				(*571*) (*ALL 571 AND SUBS*)
					OR ((Model_ID=7)
						(*AND Part_Present1 AND Part_Present2 AND Part_Present3
						AND Part_Present4 AND Part_Present5 AND Part_Present6
						AND Part_Present7 AND NOT Part_Present8 AND NOT Part_Present9
						AND NOT Part_Present10 AND NOT Part_Present11 AND NOT Part_Present12
						AND NOT Part_Present13 AND Part_Present15 AND NOT Part_Present16 
						AND NOT Part_Present17 AND NOT Part_Present18 AND NOT Part_Present19 
						AND NOT Part_Present20 AND NOT Part_Present21 AND Part_Present22 
						AND Part_Present23 AND Part_Present24 AND NOT Part_Present25 
						AND NOT Part_Present29 
						AND NOT Part_Present30 AND NOT Part_Present31 AND NOT Part_Present32 
						AND Part_Present33 AND Part_Present34 AND Part_Present35 
						AND Part_Present36 AND Part_Present37 AND Part_Present38 
						AND NOT Part_Present39 AND NOT Part_Present40 AND NOT Part_Present41 
						AND NOT Part_Present42 AND NOT Part_Present43 AND Part_Present45
						AND Part_Present46 AND Part_Present47 AND Part_Present48
						AND Part_Present49 AND Part_Present50 AND Part_Present51
						AND NOT Part_Present52 AND NOT Part_Present53 AND NOT Part_Present54
						AND NOT Part_Present55 AND NOT Part_Present56 AND NOT Part_Present57
						AND Part_Present62 AND Part_Present63 AND Part_Present64*)

						AND Part_Present1 AND Part_Present2 AND  Part_Present3
						AND Part_Present4 AND Part_Present5 AND Part_Present6
						AND Part_Present7 AND NOT Part_Present8 AND NOT Part_Present9
						AND NOT Part_Present10 AND NOT Part_Present11 AND NOT Part_Present12
						AND NOT Part_Present13 AND NOT Part_Present14 AND Part_Present15
						AND NOT Part_Present16 AND NOT Part_Present17 AND NOT Part_Present18
						AND NOT Part_Present19 AND NOT Part_Present20 AND NOT Part_Present21
						AND Part_Present22 AND Part_Present23 AND Part_Present24
						AND NOT Part_Present25 AND NOT Part_Present26 AND NOT Part_Present27
						AND NOT Part_Present28 AND NOT Part_Present29 AND NOT Part_Present30
						AND NOT Part_Present31 AND NOT Part_Present32 AND Part_Present33
						AND Part_Present34 AND Part_Present35 AND Part_Present36
						AND Part_Present37 AND Part_Present38 AND NOT Part_Present39
						AND NOT Part_Present40 AND NOT Part_Present41 AND NOT Part_Present42 
						AND NOT Part_Present43 AND NOT Part_Present44 AND Part_Present45
						AND Part_Present46 AND Part_Present47 AND Part_Present48
						AND Part_Present49 AND Part_Present50 AND Part_Present51
						AND NOT Part_Present52 AND NOT Part_Present53 AND NOT Part_Present54
						AND NOT Part_Present55 AND NOT Part_Present56 AND NOT Part_Present57
						AND NOT Part_Present58 AND NOT Part_Present59 AND NOT Part_Present60
						AND NOT Part_Present61 AND Part_Present62 AND Part_Present63
						AND Part_Present64 AND NOT Part_Present65 AND NOT Part_Present66
						AND NOT Part_Present67 AND NOT Part_Present68 AND NOT Part_Present69
						AND NOT Part_Present70 AND NOT Part_Present71 AND NOT Part_Present72
						AND NOT Part_Present73 AND NOT Part_Present74 AND NOT Part_Present75
						AND NOT Part_Present76)			
					) OR (All_Sensors_Off AND Dry_Cycle)
					
					(*504 SUBS 1,2*)
					OR (((Model_ID=8) AND All_Sensors_On.9 AND All_Sensors_On.10)							

					(*524 SUBS 1,2*)
					OR ((Model_ID=9) AND All_Sensors_On.9 AND All_Sensors_On.10)							

					(*543 SUBS 1,2,5*)
					OR ((Model_ID=10) AND All_Sensors_On.9 AND All_Sensors_On.10 AND All_Sensors_On.13)							
							
					(*526 SUBS 1-3*)
					OR ((Model_ID=11) AND All_Sensors_On.9 AND All_Sensors_On.10 AND All_Sensors_On.11)
							
					(*526 SUBS 4 ONLY*)
					OR ((Model_ID=15) AND All_Sensors_On.12)
							
					(*526 SUBS 1-4*)
					OR ((Model_ID=19) AND All_Sensors_On.9 AND All_Sensors_On.10 AND All_Sensors_On.11 AND All_Sensors_On.12)
					
					(*536 SUBS 1-3*)
					OR ((Model_ID=12) AND All_Sensors_On.9 AND All_Sensors_On.10 AND All_Sensors_On.11)
							
					(*536 SUBS 4 ONLY*)
					OR ((Model_ID=16) AND All_Sensors_On.12)
							
					(*536 SUBS 1-4*)
					OR ((Model_ID=20) AND All_Sensors_On.9 AND All_Sensors_On.10 AND All_Sensors_On.11 AND All_Sensors_On.12)
					
					(*550 SUBS 1-3*)
					OR ((Model_ID=13) AND All_Sensors_On.9 AND All_Sensors_On.10 AND All_Sensors_On.11)
							
					(*550 SUBS 4 ONLY*)
					OR ((Model_ID=17) AND All_Sensors_On.12)
							
					(*550 SUBS 1-4*)
					OR ((Model_ID=21) AND All_Sensors_On.9 AND All_Sensors_On.10 AND All_Sensors_On.11 AND All_Sensors_On.12)
					
					(*571 SUBS 1-3*)
					OR ((Model_ID=14) AND All_Sensors_On.9 AND All_Sensors_On.10 AND All_Sensors_On.11)
							
					(*571 SUBS 4 ONLY*)
					OR ((Model_ID=18) AND All_Sensors_On.12)
							
					(*571 SUBS 1-4*)
					OR ((Model_ID=22) AND All_Sensors_On.9 AND All_Sensors_On.10 AND All_Sensors_On.11 AND All_Sensors_On.12));

	(*Sensors Required for Resetting Subs*)
	(*SUB 1 - Not Checking Sub 1,2 sensors as we are building 1-3*)
	All_Sensors_On.9:= ((*NOT Part_Present1 AND NOT Part_Present2 AND NOT  Part_Present3
						AND NOT Part_Present4 AND NOT Part_Present5 AND NOT Part_Present6
						AND NOT Part_Present7*)NOT Part_Present8 AND NOT Part_Present9
						AND NOT Part_Present10 AND NOT Part_Present11 AND NOT Part_Present12
						AND NOT Part_Present13 AND NOT Part_Present14 AND NOT Part_Present15
						AND NOT Part_Present16 AND NOT Part_Present17 AND NOT Part_Present18
						AND NOT Part_Present19 AND NOT Part_Present20 (*AND NOT Part_Present21*)
						AND NOT Part_Present22 AND NOT Part_Present23 AND NOT Part_Present24
						AND NOT Part_Present25 AND NOT Part_Present26 AND NOT Part_Present27
						AND NOT Part_Present28 AND NOT Part_Present29 AND NOT Part_Present30
						AND NOT Part_Present31 AND NOT Part_Present32 AND NOT Part_Present33
						AND NOT Part_Present34 AND NOT Part_Present35 AND NOT Part_Present36
						AND NOT Part_Present37 AND NOT Part_Present38 AND NOT Part_Present39
						AND NOT Part_Present40 AND NOT Part_Present41 AND NOT Part_Present42 
						AND NOT Part_Present43 AND NOT Part_Present44 (*AND NOT Part_Present45
						AND NOT Part_Present46 AND NOT Part_Present47 AND NOT Part_Present48
						AND NOT Part_Present49 AND NOT Part_Present50 AND NOT Part_Present51*)
						AND NOT Part_Present52 AND NOT Part_Present53 AND NOT Part_Present54
						AND NOT Part_Present55 AND NOT Part_Present56 AND NOT Part_Present57
						AND NOT Part_Present58 AND NOT Part_Present59 AND NOT Part_Present60
						AND NOT Part_Present61 AND NOT Part_Present62 AND NOT Part_Present63
						AND NOT Part_Present64 AND NOT Part_Present65 AND NOT Part_Present66
						AND NOT Part_Present67 AND NOT Part_Present68 AND NOT Part_Present69
						AND NOT Part_Present70 AND NOT Part_Present71 AND NOT Part_Present72
						(*AND NOT Part_Present73*) AND NOT Part_Present74 (*AND NOT Part_Present75*)
						AND NOT Part_Present76)
					  AND
						(((Model_ID=8) AND( NOT Part_Present1 AND NOT Part_Present2 AND NOT Part_Present3
									   AND NOT Part_Present4 AND NOT Part_Present5 AND Part_Present6
									   AND Part_Present7))
										
					  OR ((Model_ID=9) AND( NOT Part_Present1 AND NOT Part_Present2 AND NOT Part_Present3
									   AND NOT Part_Present4 AND Part_Present5 AND Part_Present6
									   AND Part_Present7))
										
					  OR ((Model_ID=10) AND( NOT Part_Present1 AND NOT Part_Present2 AND NOT Part_Present3
									    AND NOT Part_Present4 AND NOT Part_Present5 AND NOT Part_Present6
									    AND Part_Present7))
									   
					  OR ((Model_ID=11) AND(Part_Present1 AND NOT Part_Present2 AND NOT Part_Present3
									    AND NOT Part_Present4 AND Part_Present5 AND Part_Present6
									    AND Part_Present7))
									   
					  OR ((Model_ID=12) AND(Part_Present1 AND NOT Part_Present2 AND NOT Part_Present3
									    AND Part_Present4 AND Part_Present5 AND Part_Present6
									    AND Part_Present7))
									   
					  OR ((Model_ID=13) AND(Part_Present1 AND NOT Part_Present2 AND Part_Present3
									    AND Part_Present4 AND Part_Present5 AND Part_Present6
									    AND Part_Present7))
									   
					  OR ((Model_ID=14) AND(Part_Present1 AND Part_Present2 AND Part_Present3
									    AND Part_Present4 AND Part_Present5 AND Part_Present6
									    AND Part_Present7)))

						OR (All_Sensors_Off AND Dry_Cycle);

	(*SUB 2 - Not Checking Sub 1,2 as we are building 1-3*)
	All_Sensors_On.10:= ((*NOT Part_Present1 AND NOT Part_Present2 AND NOT  Part_Present3
						AND NOT Part_Present4 AND NOT Part_Present5 AND NOT Part_Present6
						AND NOT Part_Present7*)NOT Part_Present8 AND NOT Part_Present9
						AND NOT Part_Present10 AND NOT Part_Present11 AND NOT Part_Present12
						AND NOT Part_Present13 AND NOT Part_Present14 AND NOT Part_Present15
						AND NOT Part_Present16 AND NOT Part_Present17 AND NOT Part_Present18
						AND NOT Part_Present19 AND NOT Part_Present20 (*AND NOT Part_Present21*)
						AND NOT Part_Present22 AND NOT Part_Present23 AND NOT Part_Present24
						AND NOT Part_Present25 AND NOT Part_Present26 AND NOT Part_Present27
						AND NOT Part_Present28 AND NOT Part_Present29 AND NOT Part_Present30
						AND NOT Part_Present31 AND NOT Part_Present32 AND NOT Part_Present33
						AND NOT Part_Present34 AND NOT Part_Present35 AND NOT Part_Present36
						AND NOT Part_Present37 AND NOT Part_Present38 AND NOT Part_Present39
						AND NOT Part_Present40 AND NOT Part_Present41 AND NOT Part_Present42 
						AND NOT Part_Present43 AND NOT Part_Present44 (*AND NOT Part_Present45
						AND NOT Part_Present46 AND NOT Part_Present47 AND NOT Part_Present48
						AND NOT Part_Present49 AND NOT Part_Present50 AND NOT Part_Present51*)
						AND NOT Part_Present52 AND NOT Part_Present53 AND NOT Part_Present54
						AND NOT Part_Present55 AND NOT Part_Present56 AND NOT Part_Present57
						AND NOT Part_Present58 AND NOT Part_Present59 AND NOT Part_Present60
						AND NOT Part_Present61 AND NOT Part_Present62 AND NOT Part_Present63
						AND NOT Part_Present64 AND NOT Part_Present65 AND NOT Part_Present66
						AND NOT Part_Present67 AND NOT Part_Present68 AND NOT Part_Present69
						AND NOT Part_Present70 AND NOT Part_Present71 AND NOT Part_Present72
						(*AND NOT Part_Present73*) AND NOT Part_Present74 (*AND NOT Part_Present75*)
						AND NOT Part_Present76)
						AND
						(((Model_ID=8) AND( NOT Part_Present45
											AND NOT Part_Present46 AND NOT Part_Present47 AND NOT Part_Present48
											AND NOT Part_Present49 AND Part_Present50 AND Part_Present51))
										
					  OR ((Model_ID=9) AND( NOT Part_Present45
											AND NOT Part_Present46 AND NOT Part_Present47 AND NOT Part_Present48
											AND Part_Present49 AND Part_Present50 AND Part_Present51))
										
					  OR ((Model_ID=10) AND( NOT Part_Present45
											AND NOT Part_Present46 AND NOT Part_Present47 AND NOT Part_Present48
											AND NOT Part_Present49 AND NOT Part_Present50 AND Part_Present51))
									   
					  OR ((Model_ID=11) AND(NOT Part_Present45
											AND NOT Part_Present46 AND NOT Part_Present47 AND Part_Present48
											AND Part_Present49 AND Part_Present50 AND Part_Present51))
									   
					  OR ((Model_ID=12) AND(NOT Part_Present45
											AND NOT Part_Present46 AND Part_Present47 AND Part_Present48
											AND Part_Present49 AND Part_Present50 AND Part_Present51))
									   
					  OR ((Model_ID=13) AND(NOT Part_Present45
											AND Part_Present46 AND Part_Present47 AND Part_Present48
											AND Part_Present49 AND Part_Present50 AND Part_Present51))
									   
					  OR ((Model_ID=14) AND(Part_Present45
											AND Part_Present46 AND Part_Present47 AND Part_Present48
											AND Part_Present49 AND Part_Present50 AND Part_Present51)))

			 OR (All_Sensors_Off AND Dry_Cycle);

	(*SUB 3 - Not Checking Sub 1,2 as we are building 1-3*)
	All_Sensors_On.11:=((*NOT Part_Present1 AND NOT Part_Present2 AND NOT  Part_Present3
						AND NOT Part_Present4 AND NOT Part_Present5 AND NOT Part_Present6
						AND NOT Part_Present7*)NOT Part_Present8 AND NOT Part_Present9
						AND NOT Part_Present10 AND NOT Part_Present11 AND NOT Part_Present12
						AND NOT Part_Present13 AND NOT Part_Present14 AND NOT Part_Present15
						AND NOT Part_Present16 AND NOT Part_Present17 AND NOT Part_Present18
						AND NOT Part_Present19 AND NOT Part_Present20 (*AND NOT Part_Present21*)
						AND NOT Part_Present22 AND NOT Part_Present23 AND NOT Part_Present24
						AND NOT Part_Present25 AND NOT Part_Present26 AND NOT Part_Present27
						AND NOT Part_Present28 AND NOT Part_Present29 AND NOT Part_Present30
						AND NOT Part_Present31 AND NOT Part_Present32 AND NOT Part_Present33
						AND NOT Part_Present34 AND NOT Part_Present35 AND NOT Part_Present36
						AND NOT Part_Present37 AND NOT Part_Present38 AND NOT Part_Present39
						AND NOT Part_Present40 AND NOT Part_Present41 AND NOT Part_Present42 
						AND NOT Part_Present43 AND NOT Part_Present44 (*AND NOT Part_Present45
						AND NOT Part_Present46 AND NOT Part_Present47 AND NOT Part_Present48
						AND NOT Part_Present49 AND NOT Part_Present50 AND NOT Part_Present51*)
						AND NOT Part_Present52 AND NOT Part_Present53 AND NOT Part_Present54
						AND NOT Part_Present55 AND NOT Part_Present56 AND NOT Part_Present57
						AND NOT Part_Present58 AND NOT Part_Present59 AND NOT Part_Present60
						AND NOT Part_Present61 AND NOT Part_Present62 AND NOT Part_Present63
						AND NOT Part_Present64 AND NOT Part_Present65 AND NOT Part_Present66
						AND NOT Part_Present67 AND NOT Part_Present68 AND NOT Part_Present69
						AND NOT Part_Present70 AND NOT Part_Present71 AND NOT Part_Present72
						(*AND NOT Part_Present73*) AND NOT Part_Present74 (*AND NOT Part_Present75*)
						AND NOT Part_Present76)
						AND
						(((Model_ID=11) AND(Part_Present21))
									   
					  OR ((Model_ID=12) AND(Part_Present21))
									   
					  OR ((Model_ID=13) AND(Part_Present21))
									   
					  OR ((Model_ID=14) AND(Part_Present21)))

		 	OR (All_Sensors_Off AND Dry_Cycle);

	(*SUB 4 - Checking only SUB 4 Sensors*)
	All_Sensors_On.12:=(NOT Part_Present1 AND NOT Part_Present2 AND NOT  Part_Present3
						AND NOT Part_Present4 AND NOT Part_Present5 AND NOT Part_Present6
						AND NOT Part_Present7  AND NOT Part_Present8 AND NOT Part_Present9
						AND NOT Part_Present10 AND NOT Part_Present11 AND NOT Part_Present12
						AND NOT Part_Present13 AND NOT Part_Present14 AND NOT Part_Present15
						AND NOT Part_Present16 AND NOT Part_Present17 AND NOT Part_Present18
						AND NOT Part_Present19 AND NOT Part_Present20 AND NOT Part_Present21
						AND NOT Part_Present22 AND NOT Part_Present23 AND NOT Part_Present24
						AND NOT Part_Present25 AND NOT Part_Present26 AND NOT Part_Present27
						AND NOT Part_Present28 AND NOT Part_Present29 AND NOT Part_Present30
						AND NOT Part_Present31 AND NOT Part_Present32 (*AND NOT Part_Present33
						AND NOT Part_Present34 AND NOT Part_Present35 AND NOT Part_Present36
						AND NOT Part_Present37*) AND NOT Part_Present38 AND NOT Part_Present39
						AND NOT Part_Present40 AND NOT Part_Present41 AND NOT Part_Present42 
						AND NOT Part_Present43 AND NOT Part_Present44 AND NOT Part_Present45
						AND NOT Part_Present46 AND NOT Part_Present47 AND NOT Part_Present48
						AND NOT Part_Present49 AND NOT Part_Present50 AND NOT Part_Present51
						AND NOT Part_Present52 AND NOT Part_Present53 AND NOT Part_Present54
						AND NOT Part_Present55 AND NOT Part_Present56 AND NOT Part_Present57
						AND NOT Part_Present58 AND NOT Part_Present59 AND NOT Part_Present60
						AND NOT Part_Present61 AND NOT Part_Present62 AND NOT Part_Present63
						AND NOT Part_Present64 AND NOT Part_Present65 AND NOT Part_Present66
						AND NOT Part_Present67 AND NOT Part_Present68 AND NOT Part_Present69
						AND NOT Part_Present70 AND NOT Part_Present71 AND NOT Part_Present72
						AND NOT Part_Present73 AND NOT Part_Present74 AND NOT Part_Present75
						AND NOT Part_Present76)
						AND
						(((Model_ID=15) AND(NOT Part_Present33
										AND NOT Part_Present34 AND NOT Part_Present35 AND Part_Present36
										AND Part_Present37))
									   
					  OR ((Model_ID=16) AND(NOT Part_Present33
										AND NOT Part_Present34 AND Part_Present35 AND Part_Present36
										AND Part_Present37))
									   
					  OR ((Model_ID=17) AND(NOT Part_Present33
										AND Part_Present34 AND Part_Present35 AND Part_Present36
										AND Part_Present37))
									   
					  OR ((Model_ID=18) AND(Part_Present33
										AND Part_Present34 AND Part_Present35 AND Part_Present36
										AND Part_Present37)))

		 	OR (All_Sensors_Off AND Dry_Cycle);
	
	(*SUB 5 - Not Checking SUB 1,2 Sensors as we build 543 SUB 5 with SUB 1,2*)
	All_Sensors_On.13:=((*NOT Part_Present1 AND NOT Part_Present2 AND NOT  Part_Present3
						AND NOT Part_Present4 AND NOT Part_Present5 AND NOT Part_Present6
						AND NOT Part_Present7  AND*) NOT Part_Present8 AND NOT Part_Present9
						AND NOT Part_Present10 AND NOT Part_Present11 AND NOT Part_Present12
						AND NOT Part_Present13 AND NOT Part_Present14 AND NOT Part_Present15
						AND NOT Part_Present16 AND NOT Part_Present17 AND NOT Part_Present18
						AND NOT Part_Present19 AND NOT Part_Present20 AND NOT Part_Present21
						AND NOT Part_Present22 AND NOT Part_Present23 AND NOT Part_Present24
						AND NOT Part_Present25 AND NOT Part_Present26 AND NOT Part_Present27
						AND NOT Part_Present28 AND NOT Part_Present29 AND NOT Part_Present30
						AND NOT Part_Present31 AND NOT Part_Present32 AND NOT Part_Present33
						AND NOT Part_Present34 AND NOT Part_Present35 AND NOT Part_Present36
						AND NOT Part_Present37 AND NOT Part_Present38 AND NOT Part_Present39
						AND NOT Part_Present40 AND NOT Part_Present41 AND NOT Part_Present42 
						AND NOT Part_Present43 AND NOT Part_Present44 (*AND NOT Part_Present45
						AND NOT Part_Present46 AND NOT Part_Present47 AND NOT Part_Present48
						AND NOT Part_Present49 AND NOT Part_Present50 AND NOT Part_Present51*)
						AND NOT Part_Present52 AND NOT Part_Present53 AND NOT Part_Present54
						AND NOT Part_Present55 AND NOT Part_Present56 AND NOT Part_Present57
						AND NOT Part_Present58 AND NOT Part_Present59 AND NOT Part_Present60
						AND NOT Part_Present61 AND NOT Part_Present62 AND NOT Part_Present63
						AND NOT Part_Present64 AND NOT Part_Present65 AND NOT Part_Present66
						AND NOT Part_Present67 AND NOT Part_Present68 AND NOT Part_Present69
						AND NOT Part_Present70 AND NOT Part_Present71 AND NOT Part_Present72
						(*AND NOT Part_Present73*) AND NOT Part_Present74 (*AND NOT Part_Present75*)
						AND NOT Part_Present76)
						AND
						(((Model_ID=10) AND(Part_Present73 AND Part_Present75)))
	
		 	OR (All_Sensors_Off AND Dry_Cycle);






















(*end*)
END_ACTION

METHOD PRIVATE Blank_NodeLayout : BOOL
VAR_INPUT
	Start_Array_Member: UINT;
END_VAR

VAR
	Index: UINT;
END_VAR
IF Start_Array_Member >=34 AND Start_Array_Member < 45 THEN
	FOR Index:= Start_Array_Member TO 45 BY 1 DO
		Discrete_Image.NodeLayout.NodeName[index]:='';
		Discrete_Image.NodeLayout.NodeType[index]:='';
		Discrete_Image.NodeState[index]:= 0;
	END_FOR

END_IF
END_METHOD

ACTION Cylinders:

(* -----------------------------------------------------------------------------------*)
(*Below are Examples only, each will have to be customized for your application
	Notes:
	- Use SODGxx-SSCC61x-xxxxxxx_Fix IO and Seq.xlsx document to capture Clamp / Cylinder I/O Layout
	- CLFaults1 thru 4 can be used to group cylinder type faults (All Clamps on CLFaults1, all Pins on CLFaults2)
		OR
	- CLFaults 1 thru 4 can be used to group cylinder UI screens 
		(All items on Cylinder_1.content screen are on CLFaults1, all items on Cylinder_2.content screen are on CLFaults2 as example)
*)
(* -----------------------------------------------------------------------------------*)

(*Clamps*)(*Clamps*)(*Clamps*)
(*Clamps*)(*Clamps*)(*Clamps*)
(*Clamps*)(*Clamps*)(*Clamps*)

		(*Clamp1*)
		Clamp1FB(
			Retracted_Sensor:= N09.I.0,
			Advanced_Sensor:= N09.I.1,
			Retract_Solenoid:= N100.Q.1,
			Advance_Solenoid:= N100.Q.0,
			Ret_Delay:= T#0.1S,
			Adv_Delay:= T#0.1S,
			Fault_Delay:= T#3.0S,
			Disable_Fault:= FALSE,
			In_Retracted_Position=> Clamp1RETD,
			In_Advanced_Position=> Clamp1ADVD,
			Faulted=> CLFaults1.1 );

		(*Clamp2*)
		Clamp2FB(
			Retracted_Sensor:= N09.I.2,
			Advanced_Sensor:= N09.I.3,
			Retract_Solenoid:= N100.Q.1 ,
			Advance_Solenoid:= N100.Q.0 ,
			Ret_Delay:= T#0.1S,
			Adv_Delay:= T#0.1S,
			Fault_Delay:= T#3.0S,
			Disable_Fault:= FALSE,
			In_Retracted_Position=> Clamp2RETD,
			In_Advanced_Position=> Clamp2ADVD,
			Faulted=> CLFaults1.2 );

		(*Clamp3*)
		Clamp3FB(
			Retracted_Sensor:= N09.I.4,
			Advanced_Sensor:= N09.I.5,
			Retract_Solenoid:= N100.Q.7,
			Advance_Solenoid:= N100.Q.6,
			Ret_Delay:= T#0.1S,
			Adv_Delay:= T#0.1S,
			Fault_Delay:= T#3.0S,
			Disable_Fault:= FALSE,
			In_Retracted_Position=> Clamp3RETD,
			In_Advanced_Position=> Clamp3ADVD,
			Faulted=> CLFaults1.3 );

		(*Clamp4*)
		Clamp4FB(
			Retracted_Sensor:= N09.I.6,
			Advanced_Sensor:= N09.I.7,
			Retract_Solenoid:= N100.Q.9,
			Advance_Solenoid:= N100.Q.8,
			Ret_Delay:= T#0.1S,
			Adv_Delay:= T#0.1S,
			Fault_Delay:= T#3.0S,
			Disable_Fault:= FALSE,
			In_Retracted_Position=> Clamp4RETD,
			In_Advanced_Position=> Clamp4ADVD,
			Faulted=> CLFaults1.4 );

		(*Clamp5*)
		Clamp5FB(
			Retracted_Sensor:= N10.I.0,
			Advanced_Sensor:= N10.I.1,
			Retract_Solenoid:= N100.Q.31,
			Advance_Solenoid:= N100.Q.30,
			Ret_Delay:= T#0.1S,
			Adv_Delay:= T#0.1S,
			Fault_Delay:= T#3.0S,
			Disable_Fault:= FALSE,
			In_Retracted_Position=> Clamp5RETD,
			In_Advanced_Position=> Clamp5ADVD,
			Faulted=> CLFaults1.5 );

		(*Clamp6*)
		Clamp6FB(
			Retracted_Sensor:= N10.I.2,
			Advanced_Sensor:= N10.I.3,
			Retract_Solenoid:= N100.Q.11,
			Advance_Solenoid:= N100.Q.10,
			Ret_Delay:= T#0.1S,
			Adv_Delay:= T#0.1S,
			Fault_Delay:= T#3.0S,
			Disable_Fault:= FALSE,
			In_Retracted_Position=> Clamp6RETD,
			In_Advanced_Position=> Clamp6ADVD,
			Faulted=> CLFaults1.6 );

		(*Clamp7*)
		Clamp7FB(
			Retracted_Sensor:= N10.I.4,
			Advanced_Sensor:= N10.I.5,
			Retract_Solenoid:= N100.Q.13,
			Advance_Solenoid:= N100.Q.12,
			Ret_Delay:= T#0.1S,
			Adv_Delay:= T#0.1S,
			Fault_Delay:= T#3.0S,
			Disable_Fault:= FALSE,
			In_Retracted_Position=> Clamp7RETD,
			In_Advanced_Position=> Clamp7ADVD,
			Faulted=> CLFaults1.7 );

		(*Clamp8*)
		Clamp8FB(
			Retracted_Sensor:= N10.I.6,
			Advanced_Sensor:= N10.I.7,
			Retract_Solenoid:= N101.Q.7,
			Advance_Solenoid:= N101.Q.6,
			Ret_Delay:= T#0.1S,
			Adv_Delay:= T#0.1S,
			Fault_Delay:= T#3.0S,
			Disable_Fault:= FALSE,
			In_Retracted_Position=> Clamp8RETD,
			In_Advanced_Position=> Clamp8ADVD,
			Faulted=> CLFaults1.8 );

		(*Clamp9*)
		Clamp9FB(
			Retracted_Sensor:= N11.I.0,
			Advanced_Sensor:= N11.I.1,
			Retract_Solenoid:= N100.Q.11,
			Advance_Solenoid:= N100.Q.10,
			Ret_Delay:= T#0.1S,
			Adv_Delay:= T#0.1S,
			Fault_Delay:= T#3.0S,
			Disable_Fault:= FALSE,
			In_Retracted_Position=> Clamp9RETD,
			In_Advanced_Position=> Clamp9ADVD,
			Faulted=> CLFaults1.9 );

		(*Clamp10*)
		Clamp10FB(
			Retracted_Sensor:= N11.I.2,
			Advanced_Sensor:= N11.I.3,
			Retract_Solenoid:= N101.Q.9,
			Advance_Solenoid:= N101.Q.8,
			Ret_Delay:= T#0.1S,
			Adv_Delay:= T#0.1S,
			Fault_Delay:= T#3.0S,
			Disable_Fault:= FALSE,
			In_Retracted_Position=> Clamp10RETD,
			In_Advanced_Position=> Clamp10ADVD,
			Faulted=> CLFaults1.10 );

		(*Clamp11*)
		Clamp11FB(
			Retracted_Sensor:= N11.I.4,
			Advanced_Sensor:= N11.I.5,
			Retract_Solenoid:= N100.Q.9,
			Advance_Solenoid:= N100.Q.8,
			Ret_Delay:= T#0.1S,
			Adv_Delay:= T#0.1S,
			Fault_Delay:= T#3.0S,
			Disable_Fault:= FALSE,
			In_Retracted_Position=> Clamp11RETD,
			In_Advanced_Position=> Clamp11ADVD,
			Faulted=> CLFaults1.11 );

		(*Clamp12*)
		Clamp12FB(
			Retracted_Sensor:= N11.I.6,
			Advanced_Sensor:= N11.I.7,
			Retract_Solenoid:= N100.Q.7,
			Advance_Solenoid:= N100.Q.6,
			Ret_Delay:= T#0.1S,
			Adv_Delay:= T#0.1S,
			Fault_Delay:= T#3.0S,
			Disable_Fault:= FALSE,
			In_Retracted_Position=> Clamp12RETD,
			In_Advanced_Position=> Clamp12ADVD,
			Faulted=> CLFaults1.12 );

		(*Clamp13*)
		Clamp13FB(
			Retracted_Sensor:= N12.I.0,
			Advanced_Sensor:= N12.I.1,
			Retract_Solenoid:= N100.Q.3,
			Advance_Solenoid:= N100.Q.2,
			Ret_Delay:= T#0.1S,
			Adv_Delay:= T#0.1S,
			Fault_Delay:= T#3.0S,
			Disable_Fault:= FALSE,
			In_Retracted_Position=> Clamp13RETD,
			In_Advanced_Position=> Clamp13ADVD,
			Faulted=> CLFaults1.13 );

		(*Clamp14*)
		Clamp14FB(
			Retracted_Sensor:= N12.I.2,
			Advanced_Sensor:= N12.I.3,
			Retract_Solenoid:= N100.Q.3,
			Advance_Solenoid:= N100.Q.2,
			Ret_Delay:= T#0.1S,
			Adv_Delay:= T#0.1S,
			Fault_Delay:= T#3.0S,
			Disable_Fault:= FALSE,
			In_Retracted_Position=> Clamp14RETD,
			In_Advanced_Position=> Clamp14ADVD,
			Faulted=> CLFaults2.1 );

		(*Clamp15*)
		Clamp15FB(
			Retracted_Sensor:= N12.I.4,
			Advanced_Sensor:= N12.I.5,
			Retract_Solenoid:= N100.Q.3,
			Advance_Solenoid:= N100.Q.2,
			Ret_Delay:= T#0.1S,
			Adv_Delay:= T#0.1S,
			Fault_Delay:= T#3.0S,
			Disable_Fault:= FALSE,
			In_Retracted_Position=> Clamp15RETD,
			In_Advanced_Position=> Clamp15ADVD,
			Faulted=> CLFaults2.2 );

		(*Clamp16*)
		Clamp16FB(
			Retracted_Sensor:= N12.I.6,
			Advanced_Sensor:= N12.I.7,
			Retract_Solenoid:= N100.Q.5,
			Advance_Solenoid:= N100.Q.4,
			Ret_Delay:= T#0.1S,
			Adv_Delay:= T#0.1S,
			Fault_Delay:= T#3.0S,
			Disable_Fault:= FALSE,
			In_Retracted_Position=> Clamp16RETD,
			In_Advanced_Position=> Clamp16ADVD,
			Faulted=> CLFaults2.3 );

		(*Clamp17*)
		Clamp17FB(
			Retracted_Sensor:= N13.I.0,
			Advanced_Sensor:= N13.I.1,
			Retract_Solenoid:= N100.Q.5,
			Advance_Solenoid:= N100.Q.4,
			Ret_Delay:= T#0.1S,
			Adv_Delay:= T#0.1S,
			Fault_Delay:= T#3.0S,
			Disable_Fault:= FALSE,
			In_Retracted_Position=> Clamp17RETD,
			In_Advanced_Position=> Clamp17ADVD,
			Faulted=> CLFaults2.4 );

		(*Clamp18*)
		Clamp18FB(
			Retracted_Sensor:= N13.I.2,
			Advanced_Sensor:= N13.I.3,
			Retract_Solenoid:= N100.Q.5,
			Advance_Solenoid:= N100.Q.4,
			Ret_Delay:= T#0.1S,
			Adv_Delay:= T#0.1S,
			Fault_Delay:= T#3.0S,
			Disable_Fault:= FALSE,
			In_Retracted_Position=> Clamp18RETD,
			In_Advanced_Position=> Clamp18ADVD,
			Faulted=> CLFaults2.5 );

		(*Clamp19*)
		Clamp19FB(
			Retracted_Sensor:= N13.I.4,
			Advanced_Sensor:= N13.I.5,
			Retract_Solenoid:= N100.Q.5,
			Advance_Solenoid:= N100.Q.4,
			Ret_Delay:= T#0.1S,
			Adv_Delay:= T#0.1S,
			Fault_Delay:= T#3.0S,
			Disable_Fault:= FALSE,
			In_Retracted_Position=> Clamp19RETD,
			In_Advanced_Position=> Clamp19ADVD,
			Faulted=> CLFaults2.6 );

		(*Clamp20*)
		Clamp20FB(
			Retracted_Sensor:= N13.I.6,
			Advanced_Sensor:= N13.I.7,
			Retract_Solenoid:= N100.Q.7,
			Advance_Solenoid:= N100.Q.6,
			Ret_Delay:= T#0.1S,
			Adv_Delay:= T#0.1S,
			Fault_Delay:= T#3.0S,
			Disable_Fault:= FALSE,
			In_Retracted_Position=> Clamp20RETD,
			In_Advanced_Position=> Clamp20ADVD,
			Faulted=> CLFaults2.7 );

		(*Clamp21*) (*TLK Changed WAS on Valve 21 Actual Piped on Valve 5*)
		Clamp21FB(
			Retracted_Sensor:= N14.I.0,
			Advanced_Sensor:= N14.I.1,
			Retract_Solenoid:= N100.Q.9, (*TLK Changed to Valve 5 WAS Piped on Valve 5 From Supplier*)
			Advance_Solenoid:= N100.Q.8, (*TLK Changed to Valve 5 WAS Piped on Valve 5 From Supplier*)
			Ret_Delay:= T#0.1S,
			Adv_Delay:= T#0.1S,
			Fault_Delay:= T#3.0S,
			Disable_Fault:= FALSE,
			In_Retracted_Position=> Clamp21RETD,
			In_Advanced_Position=> Clamp21ADVD,
			Faulted=> CLFaults2.8 );

		(*Clamp22*)
		Clamp22FB(
			Retracted_Sensor:= N14.I.2,
			Advanced_Sensor:= N14.I.3,
			Retract_Solenoid:= N100.Q.15,
			Advance_Solenoid:= N100.Q.14,
			Ret_Delay:= T#0.1S,
			Adv_Delay:= T#0.1S,
			Fault_Delay:= T#3.0S,
			Disable_Fault:= FALSE,
			In_Retracted_Position=> Clamp22RETD,
			In_Advanced_Position=> Clamp22ADVD,
			Faulted=> CLFaults2.9 );

		(*Clamp23*)
		Clamp23FB(
			Retracted_Sensor:= N14.I.4,
			Advanced_Sensor:= N14.I.5,
			Retract_Solenoid:= N100.Q.17,
			Advance_Solenoid:= N100.Q.16,
			Ret_Delay:= T#0.1S,
			Adv_Delay:= T#0.1S,
			Fault_Delay:= T#3.0S,
			Disable_Fault:= FALSE,
			In_Retracted_Position=> Clamp23RETD,
			In_Advanced_Position=> Clamp23ADVD,
			Faulted=> CLFaults2.10 );

		(*Clamp24*)
		Clamp24FB(
			Retracted_Sensor:= N14.I.6,
			Advanced_Sensor:= N14.I.7,
			Retract_Solenoid:= N101.Q.7,
			Advance_Solenoid:= N101.Q.6,
			Ret_Delay:= T#0.1S,
			Adv_Delay:= T#0.1S,
			Fault_Delay:= T#3.0S,
			Disable_Fault:= FALSE,
			In_Retracted_Position=> Clamp24RETD,
			In_Advanced_Position=> Clamp24ADVD,
			Faulted=> CLFaults2.11 );

		(*Clamp25*)
		Clamp25FB(
			Retracted_Sensor:= N15.I.0,
			Advanced_Sensor:= N15.I.1,
			Retract_Solenoid:= N100.Q.17,
			Advance_Solenoid:= N100.Q.16,
			Ret_Delay:= T#0.1S,
			Adv_Delay:= T#0.1S,
			Fault_Delay:= T#3.0S,
			Disable_Fault:= FALSE,
			In_Retracted_Position=> Clamp25RETD,
			In_Advanced_Position=> Clamp25ADVD,
			Faulted=> CLFaults2.12 );

		(*Clamp26*)
		Clamp26FB(
			Retracted_Sensor:= N15.I.2,
			Advanced_Sensor:= N15.I.3,
			Retract_Solenoid:= N100.Q.15,
			Advance_Solenoid:= N100.Q.14,
			Ret_Delay:= T#0.1S,
			Adv_Delay:= T#0.1S,
			Fault_Delay:= T#3.0S,
			Disable_Fault:= FALSE,
			In_Retracted_Position=> Clamp26RETD,
			In_Advanced_Position=> Clamp26ADVD,
			Faulted=> CLFaults2.13 );

		(*Clamp27*)
		Clamp27FB(
			Retracted_Sensor:= N15.I.4,
			Advanced_Sensor:= N15.I.5,
			Retract_Solenoid:= N101.Q.9,
			Advance_Solenoid:= N101.Q.8,
			Ret_Delay:= T#0.1S,
			Adv_Delay:= T#0.1S,
			Fault_Delay:= T#3.0S,
			Disable_Fault:= FALSE,
			In_Retracted_Position=> Clamp27RETD,
			In_Advanced_Position=> Clamp27ADVD,
			Faulted=> CLFaults2.14 );

		(*Clamp28*)
		Clamp28FB(
			Retracted_Sensor:= N15.I.6,
			Advanced_Sensor:= N15.I.7,
			Retract_Solenoid:= N100.Q.7,
			Advance_Solenoid:= N100.Q.6,
			Ret_Delay:= T#0.1S,
			Adv_Delay:= T#0.1S,
			Fault_Delay:= T#3.0S,
			Disable_Fault:= FALSE,
			In_Retracted_Position=> Clamp28RETD,
			In_Advanced_Position=> Clamp28ADVD,
			Faulted=> CLFaults2.15 );

		(*Clamp29*)
		Clamp29FB(
			Retracted_Sensor:= N16.I.0,
			Advanced_Sensor:= N16.I.1,
			Retract_Solenoid:= N100.Q.9,
			Advance_Solenoid:= N100.Q.8,
			Ret_Delay:= T#0.1S,
			Adv_Delay:= T#0.1S,
			Fault_Delay:= T#3.0S,
			Disable_Fault:= FALSE,
			In_Retracted_Position=> Clamp29RETD,
			In_Advanced_Position=> Clamp29ADVD,
			Faulted=> CLFaults2.16 );

		(*Clamp30*)
		Clamp30FB(
			Retracted_Sensor:= N16.I.2,
			Advanced_Sensor:= N16.I.3,
			Retract_Solenoid:= N100.Q.11,
			Advance_Solenoid:= N100.Q.10,
			Ret_Delay:= T#0.1S,
			Adv_Delay:= T#0.1S,
			Fault_Delay:= T#3.0S,
			Disable_Fault:= FALSE,
			In_Retracted_Position=> Clamp30RETD,
			In_Advanced_Position=> Clamp30ADVD,
			Faulted=> CLFaults2.17 );

		(*Clamp31*)
		Clamp31FB(
			Retracted_Sensor:= N16.I.4,
			Advanced_Sensor:= N16.I.5,
			Retract_Solenoid:= N101.Q.7,
			Advance_Solenoid:= N101.Q.6,
			Ret_Delay:= T#0.1S,
			Adv_Delay:= T#0.1S,
			Fault_Delay:= T#3.0S,
			Disable_Fault:= FALSE,
			In_Retracted_Position=> Clamp31RETD,
			In_Advanced_Position=> Clamp31ADVD,
			Faulted=> CLFaults3.1 );

		(*Clamp32*)
		Clamp32FB(
			Retracted_Sensor:= N16.I.6,
			Advanced_Sensor:= N16.I.7,
			Retract_Solenoid:= N100.Q.1,
			Advance_Solenoid:= N100.Q.0,
			Ret_Delay:= T#0.1S,
			Adv_Delay:= T#0.1S,
			Fault_Delay:= T#3.0S,
			Disable_Fault:= FALSE,
			In_Retracted_Position=> Clamp32RETD,
			In_Advanced_Position=> Clamp32ADVD,
			Faulted=> CLFaults3.2 );

		(*Clamp33*)
		Clamp33FB(
			Retracted_Sensor:= N17.I.0,
			Advanced_Sensor:= N17.I.1,
			Retract_Solenoid:= N100.Q.9,
			Advance_Solenoid:= N100.Q.8,
			Ret_Delay:= T#0.1S,
			Adv_Delay:= T#0.1S,
			Fault_Delay:= T#3.0S,
			Disable_Fault:= FALSE,
			In_Retracted_Position=> Clamp33RETD,
			In_Advanced_Position=> Clamp33ADVD,
			Faulted=> CLFaults3.3 );

		(*Clamp34*)
		Clamp34FB(
			Retracted_Sensor:= N17.I.2,
			Advanced_Sensor:= N17.I.3,
			Retract_Solenoid:= N100.Q.7,
			Advance_Solenoid:= N100.Q.6,
			Ret_Delay:= T#0.1S,
			Adv_Delay:= T#0.1S,
			Fault_Delay:= T#3.0S,
			Disable_Fault:= FALSE,
			In_Retracted_Position=> Clamp34RETD,
			In_Advanced_Position=> Clamp34ADVD,
			Faulted=> CLFaults3.4 );

		(*Clamp35*)
		Clamp35FB(
			Retracted_Sensor:= N17.I.4,
			Advanced_Sensor:= N17.I.5,
			Retract_Solenoid:= N100.Q.13,
			Advance_Solenoid:= N100.Q.12,
			Ret_Delay:= T#0.1S,
			Adv_Delay:= T#0.1S,
			Fault_Delay:= T#3.0S,
			Disable_Fault:= FALSE,
			In_Retracted_Position=> Clamp35RETD,
			In_Advanced_Position=> Clamp35ADVD,
			Faulted=> CLFaults3.5 );

		(*Clamp36*)
		Clamp36FB(
			Retracted_Sensor:= N17.I.6,
			Advanced_Sensor:= N17.I.7,
			Retract_Solenoid:= N100.Q.11,
			Advance_Solenoid:= N100.Q.10,
			Ret_Delay:= T#0.1S,
			Adv_Delay:= T#0.1S,
			Fault_Delay:= T#3.0S,
			Disable_Fault:= FALSE,
			In_Retracted_Position=> Clamp36RETD,
			In_Advanced_Position=> Clamp36ADVD,
			Faulted=> CLFaults3.6 );

		(*Clamp37*)
		Clamp37FB(
			Retracted_Sensor:= N18.I.0,
			Advanced_Sensor:= N18.I.1,
			Retract_Solenoid:= N100.Q.1,
			Advance_Solenoid:= N100.Q.0,
			Ret_Delay:= T#0.1S,
			Adv_Delay:= T#0.1S,
			Fault_Delay:= T#3.0S,
			Disable_Fault:= FALSE,
			In_Retracted_Position=> Clamp37RETD,
			In_Advanced_Position=> Clamp37ADVD,
			Faulted=> CLFaults3.7 );

		(*Clamp38*)
		Clamp38FB(
			Retracted_Sensor:= N18.I.2,
			Advanced_Sensor:= N18.I.3,
			Retract_Solenoid:= N100.Q.31,
			Advance_Solenoid:= N100.Q.30,
			Ret_Delay:= T#0.1S,
			Adv_Delay:= T#0.1S,
			Fault_Delay:= T#3.0S,
			Disable_Fault:= FALSE,
			In_Retracted_Position=> Clamp38RETD,
			In_Advanced_Position=> Clamp38ADVD,
			Faulted=> CLFaults3.8 );

(*Pins*)(*Pins*)(*Pins*)
(*Pins*)(*Pins*)(*Pins*)
(*Pins*)(*Pins*)(*Pins*)

		(*Pin1*)
		Pin1FB(
			Retracted_Sensor:= N18.I.4,
			Advanced_Sensor:= N18.I.5,
			Retract_Solenoid:= N100.Q.29,
			Advance_Solenoid:= N100.Q.28,
			Ret_Delay:= T#0.1S,
			Adv_Delay:= T#0.1S,
			Fault_Delay:= T#3.0S,
			Disable_Fault:= FALSE,
			In_Retracted_Position=> Pin1RETD,
			In_Advanced_Position=> Pin1ADVD,
			Faulted=> CLFaults1.14 );

		(*Pin2*)
		Pin2FB(
			Retracted_Sensor:= N18.I.6,
			Advanced_Sensor:= N18.I.7,
			Retract_Solenoid:= N101.Q.5,
			Advance_Solenoid:= N101.Q.4,
			Ret_Delay:= T#0.1S,
			Adv_Delay:= T#0.1S,
			Fault_Delay:= T#3.0S,
			Disable_Fault:= FALSE,
			In_Retracted_Position=> Pin2RETD,
			In_Advanced_Position=> Pin2ADVD,
			Faulted=> CLFaults1.15 );

		(*Pin3*)
		Pin3FB(
			Retracted_Sensor:= N19.I.0,
			Advanced_Sensor:= N19.I.1,
			Retract_Solenoid:= N101.Q.3,
			Advance_Solenoid:= N101.Q.2,
			Ret_Delay:= T#0.1S,
			Adv_Delay:= T#0.1S,
			Fault_Delay:= T#3.0S,
			Disable_Fault:= FALSE,
			In_Retracted_Position=> Pin3RETD,
			In_Advanced_Position=> Pin3ADVD,
			Faulted=> CLFaults1.16 );

		(*Pin4*)
		Pin4FB(
			Retracted_Sensor:= N19.I.2,
			Advanced_Sensor:= N19.I.3,
			Retract_Solenoid:= N100.Q.29,
			Advance_Solenoid:= N100.Q.28,
			Ret_Delay:= T#0.1S,
			Adv_Delay:= T#0.1S,
			Fault_Delay:= T#3.0S,
			Disable_Fault:= FALSE,
			In_Retracted_Position=> Pin4RETD,
			In_Advanced_Position=> Pin4ADVD,
			Faulted=> CLFaults2.18 );

		(*Pin5*)
		Pin5FB(
			Retracted_Sensor:= N19.I.4,
			Advanced_Sensor:= N19.I.5,
			Retract_Solenoid:= N101.Q.5,
			Advance_Solenoid:= N101.Q.4,
			Ret_Delay:= T#0.1S,
			Adv_Delay:= T#0.1S,
			Fault_Delay:= T#3.0S,
			Disable_Fault:= FALSE,
			In_Retracted_Position=> Pin5RETD,
			In_Advanced_Position=> Pin5ADVD,
			Faulted=> CLFaults2.19 );

		(*Pin6*)
		Pin6FB(
			Retracted_Sensor:= N19.I.6,
			Advanced_Sensor:= N19.I.7,
			Retract_Solenoid:= N101.Q.3,
			Advance_Solenoid:= N101.Q.2,
			Ret_Delay:= T#0.1S,
			Adv_Delay:= T#0.1S,
			Fault_Delay:= T#3.0S,
			Disable_Fault:= FALSE,
			In_Retracted_Position=> Pin6RETD,
			In_Advanced_Position=> Pin6ADVD,
			Faulted=> CLFaults2.20 );

		(*Pin7*)
		Pin7FB(
			Retracted_Sensor:= N20.I.0,
			Advanced_Sensor:= N20.I.1,
			Retract_Solenoid:= N101.Q.5,
			Advance_Solenoid:= N101.Q.4,
			Ret_Delay:= T#0.1S,
			Adv_Delay:= T#0.1S,
			Fault_Delay:= T#3.0S,
			Disable_Fault:= FALSE,
			In_Retracted_Position=> Pin7RETD,
			In_Advanced_Position=> Pin7ADVD,
			Faulted=> CLFaults3.9 );

		(*Pin8*)
		Pin8FB(
			Retracted_Sensor:= N20.I.2,
			Advanced_Sensor:= N20.I.3,
			Retract_Solenoid:= N100.Q.29,
			Advance_Solenoid:= N100.Q.28,
			Ret_Delay:= T#0.1S,
			Adv_Delay:= T#0.1S,
			Fault_Delay:= T#3.0S,
			Disable_Fault:= FALSE,
			In_Retracted_Position=> Pin8RETD,
			In_Advanced_Position=> Pin8ADVD,
			Faulted=> CLFaults3.10 );

(*Slides*)(*Slides*)(*Slides*)
(*Slides*)(*Slides*)(*Slides*)
(*Slides*)(*Slides*)(*Slides*)

		(*Slide1*)
		Slide1FB(
			Retracted_Sensor:= N20.I.4,
			Advanced_Sensor:= N20.I.5,
			Retract_Solenoid:= N100.Q.27,
			Advance_Solenoid:= N100.Q.26,
			Adv_Delay:= T#0.2S,
			Ret_Delay:= T#0.2S,
			Fault_Delay:= T#4.0S,
			Disable_Fault:= FALSE,
			In_Retracted_Position=> Slide1RETD,
			In_Advanced_Position=> Slide1ADVD,
			Faulted=> CLFaults1.17 );

		(*Slide2*)
		Slide2FB(
			Retracted_Sensor:= N20.I.6,
			Advanced_Sensor:= N20.I.7,
			Retract_Solenoid:= N100.Q.27,
			Advance_Solenoid:= N100.Q.26,
			Adv_Delay:= T#0.2S,
			Ret_Delay:= T#0.2S,
			Fault_Delay:= T#4.0S,
			Disable_Fault:= FALSE,
			In_Retracted_Position=> Slide2RETD,
			In_Advanced_Position=> Slide2ADVD,
			Faulted=> CLFaults1.18 );

		(*Slide3*)
		Slide3FB(
			Retracted_Sensor:= N21.I.0,
			Advanced_Sensor:= N21.I.1,
			Retract_Solenoid:= N100.Q.31,
			Advance_Solenoid:= N100.Q.30,
			Adv_Delay:= T#0.2S,
			Ret_Delay:= T#0.2S,
			Fault_Delay:= T#4.0S,
			Disable_Fault:= FALSE,
			In_Retracted_Position=> Slide3RETD,
			In_Advanced_Position=> Slide3ADVD,
			Faulted=> CLFaults1.19 );

		(*Slide4*)
		Slide4FB(
			Retracted_Sensor:= N21.I.2,
			Advanced_Sensor:= N21.I.3,
			Retract_Solenoid:= N100.Q.19,
			Advance_Solenoid:= N100.Q.18,
			Adv_Delay:= T#0.2S,
			Ret_Delay:= T#0.2S,
			Fault_Delay:= T#4.0S,
			Disable_Fault:= FALSE,
			In_Retracted_Position=> Slide4RETD,
			In_Advanced_Position=> Slide4ADVD,
			Faulted=> CLFaults1.20 );

		(*Slide5*)
		Slide5FB(
			Retracted_Sensor:= N21.I.4,
			Advanced_Sensor:= N21.I.5,
			Retract_Solenoid:= N100.Q.31,
			Advance_Solenoid:= N100.Q.30,
			Adv_Delay:= T#0.2S,
			Ret_Delay:= T#0.2S,
			Fault_Delay:= T#4.0S,
			Disable_Fault:= FALSE,
			In_Retracted_Position=> Slide5RETD,
			In_Advanced_Position=> Slide5ADVD,
			Faulted=> CLFaults1.21 );

		(*Slide6*)
		Slide6FB(
			Retracted_Sensor:= N21.I.6,
			Advanced_Sensor:= N21.I.7,
			Retract_Solenoid:= N100.Q.21,
			Advance_Solenoid:= N100.Q.20,
			Adv_Delay:= T#0.2S,
			Ret_Delay:= T#0.2S,
			Fault_Delay:= T#4.0S,
			Disable_Fault:= FALSE,
			In_Retracted_Position=> Slide6RETD,
			In_Advanced_Position=> Slide6ADVD,
			Faulted=> CLFaults2.21 );

		(*Slide7*)
		Slide7FB(
			Retracted_Sensor:= N22.I.0,
			Advanced_Sensor:= N22.I.1,
			Retract_Solenoid:= N100.Q.23,
			Advance_Solenoid:= N100.Q.22,
			Adv_Delay:= T#0.2S,
			Ret_Delay:= T#0.2S,
			Fault_Delay:= T#4.0S,
			Disable_Fault:= FALSE,
			In_Retracted_Position=> Slide7RETD,
			In_Advanced_Position=> Slide7ADVD,
			Faulted=> CLFaults2.22 );

		(*Slide8*)
		Slide8FB(
			Retracted_Sensor:= N22.I.2,
			Advanced_Sensor:= N22.I.3,
			Retract_Solenoid:= N100.Q.19,
			Advance_Solenoid:= N100.Q.18,
			Adv_Delay:= T#0.2S,
			Ret_Delay:= T#0.2S,
			Fault_Delay:= T#4.0S,
			Disable_Fault:= FALSE,
			In_Retracted_Position=> Slide8RETD,
			In_Advanced_Position=> Slide8ADVD,
			Faulted=> CLFaults2.23 );

		(*Slide9*)
		Slide9FB(
			Retracted_Sensor:= N22.I.4,
			Advanced_Sensor:= N22.I.5,
			Retract_Solenoid:= N100.Q.31,
			Advance_Solenoid:= N100.Q.30,
			Adv_Delay:= T#0.2S,
			Ret_Delay:= T#0.2S,
			Fault_Delay:= T#4.0S,
			Disable_Fault:= FALSE,
			In_Retracted_Position=> Slide9RETD,
			In_Advanced_Position=> Slide9ADVD,
			Faulted=> CLFaults2.24 );

		(*Slide10*)
		Slide10FB(
			Retracted_Sensor:= N22.I.6,
			Advanced_Sensor:= N22.I.7,
			Retract_Solenoid:= N100.Q.25,
			Advance_Solenoid:= N100.Q.24,
			Adv_Delay:= T#0.2S,
			Ret_Delay:= T#0.2S,
			Fault_Delay:= T#4.0S,
			Disable_Fault:= FALSE,
			In_Retracted_Position=> Slide10RETD,
			In_Advanced_Position=> Slide10ADVD,
			Faulted=> CLFaults2.25 );		

		(*Slide11*)
		Slide11FB(
			Retracted_Sensor:= N23.I.0,
			Advanced_Sensor:= N23.I.1,
			Retract_Solenoid:= N100.Q.19,
			Advance_Solenoid:= N100.Q.18,
			Adv_Delay:= T#0.2S,
			Ret_Delay:= T#0.2S,
			Fault_Delay:= T#4.0S,
			Disable_Fault:= FALSE,
			In_Retracted_Position=> Slide11RETD,
			In_Advanced_Position=> Slide11ADVD,
			Faulted=> CLFaults2.26 );

		(*Slide12*)
		Slide12FB(
			Retracted_Sensor:= N23.I.2,
			Advanced_Sensor:= N23.I.3,
			Retract_Solenoid:= N100.Q.31,
			Advance_Solenoid:= N100.Q.30,
			Adv_Delay:= T#0.2S,
			Ret_Delay:= T#0.2S,
			Fault_Delay:= T#4.0S,
			Disable_Fault:= FALSE,
			In_Retracted_Position=> Slide12RETD,
			In_Advanced_Position=> Slide12ADVD,
			Faulted=> CLFaults2.27 );

		(*Slide13*)
		Slide13FB(
			Retracted_Sensor:= N23.I.4,
			Advanced_Sensor:= N23.I.5,
			Retract_Solenoid:= N100.Q.31,
			Advance_Solenoid:= N100.Q.30,
			Adv_Delay:= T#0.2S,
			Ret_Delay:= T#0.2S,
			Fault_Delay:= T#4.0S,
			Disable_Fault:= FALSE,
			In_Retracted_Position=> Slide13RETD,
			In_Advanced_Position=> Slide13ADVD,
			Faulted=> CLFaults3.11 );

		(*Slide14*)
		Slide14FB(
			Retracted_Sensor:= N23.I.6,
			Advanced_Sensor:= N23.I.7,
			Retract_Solenoid:= N100.Q.27,
			Advance_Solenoid:= N100.Q.26,
			Adv_Delay:= T#0.2S,
			Ret_Delay:= T#0.2S,
			Fault_Delay:= T#4.0S,
			Disable_Fault:= FALSE,
			In_Retracted_Position=> Slide14RETD,
			In_Advanced_Position=> Slide14ADVD,
			Faulted=> CLFaults3.12 );

		(*Slide15*)
		Slide15FB(
			Retracted_Sensor:= N24.I.0,
			Advanced_Sensor:= N24.I.1,
			Retract_Solenoid:= N100.Q.27,
			Advance_Solenoid:= N100.Q.26,
			Adv_Delay:= T#0.2S,
			Ret_Delay:= T#0.2S,
			Fault_Delay:= T#4.0S,
			Disable_Fault:= FALSE,
			In_Retracted_Position=> Slide15RETD,
			In_Advanced_Position=> Slide15ADVD,
			Faulted=> CLFaults3.13 );

(*QA*)(*QA*)(*QA*)
(*QA*)(*QA*)(*QA*)
(*QA*)(*QA*)(*QA*)

		(*QA Check1*)
		QACheck1FB(
			Retracted_Sensor:= N24.I.2,
			Advanced_Sensor:= N24.I.3,
			Retract_Solenoid:= N101.Q.1,
			Advance_Solenoid:= N101.Q.0,
			Ret_Delay:= T#0.1S,
			Adv_Delay:= T#0.1S,
			Fault_Delay:= T#3.0S,
			Disable_Fault:= FALSE,
			In_Retracted_Position=> QACheck1RETD,
			In_Advanced_Position=> QACheck1ADVD,
			Faulted=> CLFaults4.1 );

		(*QA Check2*)
		QACheck2FB(
			Retracted_Sensor:= N24.I.4,
			Advanced_Sensor:= N24.I.5,
			Retract_Solenoid:= N101.Q.1,
			Advance_Solenoid:= N101.Q.0,
			Ret_Delay:= T#0.1S,
			Adv_Delay:= T#0.1S,
			Fault_Delay:= T#3.0S,
			Disable_Fault:= FALSE,
			In_Retracted_Position=> QACheck2RETD,
			In_Advanced_Position=> QACheck2ADVD,
			Faulted=> CLFaults4.2 );

		(*QA Check3*)
		QACheck3FB(
			Retracted_Sensor:= N24.I.6,
			Advanced_Sensor:= N24.I.7,
			Retract_Solenoid:= N101.Q.1,
			Advance_Solenoid:= N101.Q.0,
			Ret_Delay:= T#0.1S,
			Adv_Delay:= T#0.1S,
			Fault_Delay:= T#3.0S,
			Disable_Fault:= FALSE,
			In_Retracted_Position=> QACheck3RETD,
			In_Advanced_Position=> QACheck3ADVD,
			Faulted=> CLFaults4.3 );

		(*QA Check4*)
		QACheck4FB(
			Retracted_Sensor:= N25.I.0,
			Advanced_Sensor:= N25.I.1,
			Retract_Solenoid:= N101.Q.1,
			Advance_Solenoid:= N101.Q.0,
			Ret_Delay:= T#0.1S,
			Adv_Delay:= T#0.1S,
			Fault_Delay:= T#3.0S,
			Disable_Fault:= FALSE,
			In_Retracted_Position=> QACheck4RETD,
			In_Advanced_Position=> QACheck4ADVD,
			Faulted=> CLFaults4.4 );

		(*QA Check5*)
		QACheck5FB(
			Retracted_Sensor:= N25.I.2,
			Advanced_Sensor:= N25.I.3,
			Retract_Solenoid:= N101.Q.1,
			Advance_Solenoid:= N101.Q.0,
			Ret_Delay:= T#0.1S,
			Adv_Delay:= T#0.1S,
			Fault_Delay:= T#3.0S,
			Disable_Fault:= FALSE,
			In_Retracted_Position=> QACheck5RETD,
			In_Advanced_Position=> QACheck5ADVD,
			Faulted=> CLFaults4.5 );

		(*QA Check6*)
		QACheck6FB(
			Retracted_Sensor:= N25.I.4,
			Advanced_Sensor:= N25.I.5,
			Retract_Solenoid:= N101.Q.1,
			Advance_Solenoid:= N101.Q.0,
			Ret_Delay:= T#0.1S,
			Adv_Delay:= T#0.1S,
			Fault_Delay:= T#3.0S,
			Disable_Fault:= FALSE,
			In_Retracted_Position=> QACheck6RETD,
			In_Advanced_Position=> QACheck6ADVD,
			Faulted=> CLFaults4.6 );


(*end*)
END_ACTION

ACTION Hardware:

(*Pass Node States into Array  in order on Physical Fixture*)

	NodeState:=NodeLayout.State;


(*$$$$$$$$$$$$$$$$$$$$$$$$$$$$$$$$$$$$$$$$$$$$$$$$Gather Status Of Hardware $$$$$$$$$$$$$$$$$$$$$$$$$$$$$$$$$$$$$$$$$$$$$$$$$$$$*)

	(*Sub Fixture Nodes ok*)
	IF 	(Model_ID=1 AND N32.InfoData.State=8 AND N33.InfoData.State=8) (*Model 504 (1) and Model 524(2) uses Nodes 31/32*)
			OR
		(Model_ID=2 AND N32.InfoData.State=8 AND N33.InfoData.State=8)
			OR
		(Model_ID=3 AND N42.InfoData.State=8 AND N43.InfoData.State=8) (*Model 543 (3) uses Nodes 42/43*)
			OR
		(Model_ID=4 AND N40.InfoData.State=8 AND N41.InfoData.State=8) (*Model 526 (4) uses Nodes 40/41*)
			OR
		(Model_ID=5 AND N38.InfoData.State=8 AND N39.InfoData.State=8) (*Model 536 (5) uses Nodes 38/39*)
			OR
		(Model_ID=6 AND N36.InfoData.State=8 AND N37.InfoData.State=8) (*Model 550 (6) uses Nodes 36/37*)
			OR
		(Model_ID=7 AND N34.InfoData.State=8 AND N35.InfoData.State=8) (*Model 571 (7) uses Nodes 34/35*)
		THEN
			SubNode_OK:= TRUE;
	ELSE
			SubNode_OK:= FALSE;
	END_IF;


	(*Discrete I/O Nodes*)
	IF (*(N00.InfoData.State=8 AND SubNode_OK)*) (*Fix doesn't have an EP1111*) 
		(N01.InfoData.State=8 OR (Discrete_In.Input_Node_Count<2))
		AND (N02.InfoData.State=8 OR (Discrete_In.Input_Node_Count<3))
		AND (N03.InfoData.State=8 OR (Discrete_In.Input_Node_Count<4))
		AND (N04.InfoData.State=8 OR (Discrete_In.Input_Node_Count<5))
		AND (N05.InfoData.State=8 OR (Discrete_In.Input_Node_Count<6))
		AND (N06.InfoData.State=8 OR (Discrete_In.Input_Node_Count<7))
		AND (N07.InfoData.State=8 OR (Discrete_In.Input_Node_Count<8))
		AND (N08.InfoData.State=8 OR (Discrete_In.Input_Node_Count<9))
		AND (N09.InfoData.State=8 OR (Discrete_In.Input_Node_Count<10))
		AND (N10.InfoData.State=8 OR (Discrete_In.Input_Node_Count<11))
		AND (N11.InfoData.State=8 OR (Discrete_In.Input_Node_Count<12))
		AND (N12.InfoData.State=8 OR (Discrete_In.Input_Node_Count<13))
		AND (N13.InfoData.State=8 OR (Discrete_In.Input_Node_Count<14))
		AND (N14.InfoData.State=8 OR (Discrete_In.Input_Node_Count<15))
		AND (N15.InfoData.State=8 OR (Discrete_In.Input_Node_Count<16))
		AND (N16.InfoData.State=8 OR (Discrete_In.Input_Node_Count<17))
		AND (N17.InfoData.State=8 OR (Discrete_In.Input_Node_Count<18))
		AND (N18.InfoData.State=8 OR (Discrete_In.Input_Node_Count<19))
		AND (N19.InfoData.State=8 OR (Discrete_In.Input_Node_Count<20))
		AND (N20.InfoData.State=8 OR (Discrete_In.Input_Node_Count<21))
		AND (N21.InfoData.State=8 OR (Discrete_In.Input_Node_Count<22))
		AND (N22.InfoData.State=8 OR (Discrete_In.Input_Node_Count<23))
		AND (N23.InfoData.State=8 OR (Discrete_In.Input_Node_Count<24))
		AND (N24.InfoData.State=8 OR (Discrete_In.Input_Node_Count<25))
		AND (N25.InfoData.State=8 OR (Discrete_In.Input_Node_Count<26))
		AND (N26.InfoData.State=8 OR (Discrete_In.Input_Node_Count<27))
		AND (N27.InfoData.State=8 OR (Discrete_In.Input_Node_Count<28))
		AND (N28.InfoData.State=8 OR (Discrete_In.Input_Node_Count<29))
		AND (N29.InfoData.State=8 OR (Discrete_In.Input_Node_Count<30))
		AND (N30.InfoData.State=8 OR (Discrete_In.Input_Node_Count<31))
		AND (N31.InfoData.State=8 OR (Discrete_In.Input_Node_Count<32))
		
		AND (N100_STAT.InfoData.State=8 OR (Discrete_In.VB_Node_Count<1))
		AND (N101_STAT.InfoData.State=8 OR (Discrete_In.VB_Node_Count<2))
		AND (N102_STAT.InfoData.State=8 OR (Discrete_In.VB_Node_Count<3))


		THEN
			DiscreteNode_OK:=TRUE;

	ELSE
			DiscreteNode_OK:=FALSE;

	END_IF;


	(*Cable Break Detection*)
	(*Function Returns Flags to warn of possible cable break*)
	ECatSlave_Cable_Breaks:= FUN_GTAC_EcatSlaveConnState_64bit(NodeState);			
	





















(*end*)
END_ACTION

ACTION Production:
(*$$$$$$$$$$$$$$$$$$$$$$$$$$$$$$$$$$$ Production Information $$$$$$$$$$$$$$$$$$$$$$$$$$$$$$$$$$$$$$$$$$*)
	(*Increment Production Counter*)
	Prod_Inc.CLK:= Unload_Complete;
	Prod_Inc();
	IF Prod_Inc.Q
		THEN
		Production_Count:= Production_Count+1;
	END_IF;
	IF Discrete_In.ResetProd
		THEN
		Production_Count:= 0;
	END_IF;
	Prod_Count_Out:= Production_Count;

(*~~~~~~~~~~~~~~~~~~~~~~~~~~~~~~~~Production Report~~~~~~~~~~~~~~~~~~~~~~~~~*)
	(*Input Data*)
	Production_Report.Machine_Serial:= GTAC_CONFIG.Machine_Serial;
	Production_Report.Machine_Common_Name:= GTAC_CONFIG.Machine_Common_Name;
	Production_Report.Prod_Inc:= Prod_Inc.Q;
	Production_Report.Scrap_Inc:= In_From_ICxx.QA_Request_RH;
	Production_Report.Scrap_Dec:= In_From_ICxx.QA_Reinsert_RH;
	Production_Report.Reference_TimeDate:= MAIN.Local_Time;
	Production_Report.Reference_Target_Time:= GTAC_CONFIG.ProdConfig_Target_CycleTime; 					(*This is the machine Expected Cycle Time*)
	Production_Report.Config_Day_TOD:= GTAC_CONFIG.ProdConfig_Day;										(*Pass Each Shift Configuration Structure (Start/End Time, Break Times etc*)
	Production_Report.Config_Aft_TOD:= GTAC_CONFIG.ProdConfig_Aft;
	Production_Report.Config_Mid_TOD:= GTAC_CONFIG.ProdConfig_Mid;
	Production_Report.Config_Shift_Enables:= GTAC_CONFIG.ProdConfig_Common.Shift_Enables;					(*Enable Bits for Shifts*)
	Production_Report.Config_Break_Count:= GTAC_CONFIG.ProdConfig_Common.Break_Count;						(*Select Amount of Breaks per shift*)
	Production_Report.Machine_StoppedBy_Fault:= Faults.System_Major_Fault;
	Production_Report.Enable_InShift_Change:= GTAC_CONFIG.ProdConfig_Option_SelectInShiftChange;				(*Allows Operator 5 mins at start and end of shift for clean up*)
	(*Call FB*)
	IF NOT MAIN.Starting_Scan_Pulse
		THEN
		Production_Report();
	END_IF;
	(*Output Data*)
	Out_To_ICxx.ProdReport[1].Curr_Prod_Report:= Production_Report.Shift_Report[0];
	Out_To_ICxx.ProdReport[1].Days_Prod_Report:= Production_Report.Shift_Report[1];
	Out_To_ICxx.ProdReport[1].Aft_Prod_Report:= Production_Report.Shift_Report[2];
	Out_To_ICxx.ProdReport[1].Mid_Prod_Report:= Production_Report.Shift_Report[3];

(*~~~~~~~~~~~~~~~~~~~~~~~~~~~~~~~~ Cycle Time Counters ~~~~~~~~~~~~~~~~~~~~~~~~~*)
	(*Move Previous To Register*)
	Cycle_Time_Pulse.CLK:= Unload_Complete;
	Cycle_Time_Pulse();
	IF Cycle_Time_Pulse.Q
		THEN
		PrevCycle_Time_Out:= Cycle_Time_Out;
	END_IF;
	(*Monitor Current Cycle Time (Full Cycle Time of Process)*)
		Cycle_Time.PT:= T#9999S;
		Cycle_Time.IN:= NOT Cycle_Time_Pulse.Q AND In_Auto;
		Cycle_Time();
		Cycle_Time_Out:= Cycle_Time.ET;

	(*Monitor Load Time*)
		IF In_Auto AND NOT Start_Seal_Robots AND NOT Start_Stud_Robots AND NOT Start_Weld_Robots  AND NOT Weld_Robots_Clear AND NOT Unload_Complete
			THEN
			Load_Time_Out:= Load_Time.ET;
		END_IF;
		Load_Time.PT:= T#9999S;
		Load_Time.IN:= In_Auto AND NOT Start_Seal_Robots AND NOT Start_Stud_Robots AND NOT Start_Weld_Robots  AND NOT Weld_Robots_Clear AND NOT Unload_Complete;
		Load_Time();

	(*Monitor Robot Sealing Time*)
		IF NOT Seal_Robots_Clear
			THEN
			Seal_Time_Out:= Seal_Time.ET;
		END_IF;
		Seal_Time.PT:= T#9999S;
		Seal_Time.IN:= NOT Seal_Robots_Clear;
		Seal_Time();

	(*Monitor Robot Stud Time*)
		IF NOT Stud_Robots_Clear
			THEN
			Stud_Time_Out:= Stud_Time.ET;
		END_IF;
		Stud_Time.PT:= T#9999S;
		Stud_Time.IN:= NOT Stud_Robots_Clear;
		Stud_Time();

	(*Monitor Robot Welding Time*)
		IF NOT Weld_Robots_Clear
			THEN
			Weld_Time_Out:= Weld_Time.ET;
		END_IF;
		Weld_Time.PT:= T#9999S;
		Weld_Time.IN:= NOT Weld_Robots_Clear;
		Weld_Time();

	(*Monitor Robot Turntable Time*)
		IF NOT Turntable_Clear
			THEN
			Turn_Time_Out:= Turn_Time.ET;
		END_IF;
		Turn_Time.PT:= T#9999S;
		Turn_Time.IN:= NOT Turntable_Clear;
		Turn_Time();

	(*Monitor Unload Time*)
		IF Welding_Complete
			THEN
			Unload_Time_Out:= Unload_Time.ET;
		END_IF;
		Unload_Time.PT:= T#9999S;
		Unload_Time.IN:= Welding_Complete;
		Unload_Time();

(*~~~~~~~~~~~~~~~~~~~~~~~~~~~~~~~~Product Data Report~~~~~~~~~~~~~~~~~~~~~~~~~*)
(*Can be used to load and store product specific data (pass fail results, measurements etc) into DB*)
(*Triggers to start actual storage are contained in GTAC_CONFIG.Reports*)

(*Load Data into persistent area*)
	Fix01_ProductData_Pers.Product_Model_ID:= Model_ID;
	Fix01_ProductData_Pers.Machine_Serial:= GTAC_CONFIG.Machine_Serial;
	Fix01_ProductData_Pers.Machine_Common_Name:= GTAC_CONFIG.Machine_Common_Name;
	Fix01_ProductData_Pers.Operator_ID:= 0;					(*for future*)
	Fix01_ProductData_Pers.Product_Serial:= 'NA';
	CASE Model_ID OF
		1:	Fix01_ProductData_Pers.Product_Number:= '504';
		2:	Fix01_ProductData_Pers.Product_Number:= '524';
		3:	Fix01_ProductData_Pers.Product_Number:= '543';
		4:	Fix01_ProductData_Pers.Product_Number:= '526';
		5:	Fix01_ProductData_Pers.Product_Number:= '536';
		6:	Fix01_ProductData_Pers.Product_Number:= '550';
		7:	Fix01_ProductData_Pers.Product_Number:= '571';
	END_CASE;
	Fix01_ProductData_Pers.Product_Common_Name:= 'Volvo Bumper';
		(*Build part specific data arrays, simply leave un-used elements blank (Arrays are [0..31]*)
		(*Pass / Fail Notes - Used to capture overall terms like 'Pass' 'Fail' 'NA' etc.*)	
		IF Weld_Complete_Ack THEN
			Fix01_ProductData_Pers.Generic_PassFail_Notes[1]:= 'Comp';
		END_IF;
	
	(*Transfer Product Data to UI, see MAIN.Product_Data*)		
	Out_To_ICxx.ProductReport[1]:= Fix01_ProductData_Pers;
END_ACTION

ACTION Proxies:


(*+++++++++++THIS AREA IS CUSTOM PER INSTALLATION AND WILL HAVE TO BE MODIFIED PER +++++++++++++*)
(*+++++++++++THIS AREA IS CUSTOM PER INSTALLATION AND WILL HAVE TO BE MODIFIED PER +++++++++++++*)



	(*Part 1 Present*)
		Part_Present1FB(
			Sensor_Input:= N01.I.0,
			On_Trigger1:= Enable_Motion AND In_Auto AND NOT Unload_Complete,
			On_Trigger2:= (Model_ID =4) OR (Model_ID=11) OR (Model_ID=19) OR (Model_ID =5) OR (Model_ID=12) OR (Model_ID=20)
					   OR (Model_ID=6) OR (Model_ID=13) OR (Model_ID=21) OR (Model_ID=7) OR (Model_ID=14) OR (Model_ID=22),
			Off_Trigger1:= Dry_Cycle OR (Cycle_Complete AND NOT Enable_Motion),
			Off_Trigger2:= TRUE,
			Disable_Faults:= Dry_Cycle OR (Weld_Robots_WorkingOK) OR Turntable_Bypassed,
			Fault_Delay:= T#1.5s,
			Status=> Part_Present1,
			Faulted=>  PPFaults.1);

	(*Part 2 Present*)
		Part_Present2FB(
			Sensor_Input:= N01.I.1,
			On_Trigger1:= Enable_Motion AND In_Auto AND NOT Unload_Complete,
			On_Trigger2:=  (Model_ID=7) OR (Model_ID=14) OR (Model_ID=22),
			Off_Trigger1:= Dry_Cycle OR (Cycle_Complete  AND NOT Enable_Motion),
			Off_Trigger2:= TRUE,
			Disable_Faults:= Dry_Cycle OR (Weld_Robots_WorkingOK) OR Turntable_Bypassed,
			Fault_Delay:= T#1.5s,
			Status=> Part_Present2,
			Faulted=>  PPFaults.2);

	(*Part 3 Present*)
		Part_Present3FB(
			Sensor_Input:= N01.I.2,
			On_Trigger1:= Enable_Motion AND In_Auto AND NOT Unload_Complete,
			On_Trigger2:= (Model_ID=6) OR (Model_ID=13) OR (Model_ID=21) OR (Model_ID=7) OR (Model_ID=14) OR (Model_ID=22),
			Off_Trigger1:= Dry_Cycle OR (Cycle_Complete  AND NOT Enable_Motion),
			Off_Trigger2:= TRUE,
			Disable_Faults:= Dry_Cycle OR (Weld_Robots_WorkingOK) OR Turntable_Bypassed,
			Fault_Delay:= T#1.5s,
			Status=> Part_Present3,
			Faulted=>  PPFaults.3);

	(*Part 4 Present*)
		Part_Present4FB(
			Sensor_Input:=N01.I.3,
			On_Trigger1:= Enable_Motion AND In_Auto AND NOT Unload_Complete,
			On_Trigger2:= (Model_ID =5) OR (Model_ID=12) OR (Model_ID=20) OR (Model_ID=6) OR (Model_ID=13) OR (Model_ID=21)
					   OR (Model_ID=7) OR (Model_ID=14) OR (Model_ID=22),
			Off_Trigger1:= Dry_Cycle OR (Cycle_Complete  AND NOT Enable_Motion),
			Off_Trigger2:= TRUE,
			Disable_Faults:= Dry_Cycle OR (Weld_Robots_WorkingOK) OR Turntable_Bypassed,
			Fault_Delay:= T#1.5s,
			Status=> Part_Present4,
			Faulted=>  PPFaults.4);

	(*Part 5 Present*)
		Part_Present5FB(
			Sensor_Input:= N01.I.4,
			On_Trigger1:= Enable_Motion AND In_Auto AND NOT Unload_Complete AND ((Model_ID<>3) OR (Model_ID<>10)),
			On_Trigger2:= (Model_ID =2) OR (Model_ID=9)
					   OR (Model_ID =4) OR (Model_ID=11) OR (Model_ID=19) OR (Model_ID =5) OR (Model_ID=12) OR (Model_ID=20)
					   OR (Model_ID=6) OR (Model_ID=13) OR (Model_ID=21) OR (Model_ID=7) OR (Model_ID=14) OR (Model_ID=22),
			Off_Trigger1:= Dry_Cycle OR (Cycle_Complete  AND NOT Enable_Motion),
			Off_Trigger2:= TRUE,
			Disable_Faults:= Dry_Cycle OR (Weld_Robots_WorkingOK) OR Turntable_Bypassed,
			Fault_Delay:= T#1.5s,
			Status=> Part_Present5,
			Faulted=>  PPFaults.5);

	(*Part 6 Present*)
		Part_Present6FB(
			Sensor_Input:= N01.I.5,
			On_Trigger1:= Enable_Motion AND In_Auto AND NOT Unload_Complete AND ((Model_ID<>3) OR (Model_ID<>10)),
			On_Trigger2:= (Model_ID =1) OR (Model_ID=8) OR (Model_ID =2) OR (Model_ID=9)
					   OR (Model_ID =4) OR (Model_ID=11) OR (Model_ID=19) OR (Model_ID =5) OR (Model_ID=12) OR (Model_ID=20)
					   OR (Model_ID=6) OR (Model_ID=13) OR (Model_ID=21) OR (Model_ID=7) OR (Model_ID=14) OR (Model_ID=22),
			Off_Trigger1:= Dry_Cycle OR (Cycle_Complete  AND NOT Enable_Motion),
			Off_Trigger2:= TRUE,
			Disable_Faults:= Dry_Cycle OR (Weld_Robots_WorkingOK) OR Turntable_Bypassed,
			Fault_Delay:= T#1.5s,
			Status=> Part_Present6,
			Faulted=>  PPFaults.6);

	(*Part 7 Present*)
		Part_Present7FB(
			Sensor_Input:= N01.I.6,
			On_Trigger1:= Enable_Motion AND In_Auto AND NOT Unload_Complete,
			On_Trigger2:= TRUE,
			Off_Trigger1:= Dry_Cycle OR (Cycle_Complete  AND NOT Enable_Motion),
			Off_Trigger2:= TRUE,
			Disable_Faults:= Dry_Cycle OR (Weld_Robots_WorkingOK) OR Turntable_Bypassed,
			Fault_Delay:= T#1.5s,
			Status=> Part_Present7,
			Faulted=>  PPFaults.7);

	(*Part 8 Present*)
		Part_Present8FB(
			Sensor_Input:= N01.I.7,
			On_Trigger1:= Enable_Motion AND In_Auto AND NOT Welding_Complete AND (Model_ID<>3),
			On_Trigger2:= TRUE,
			Off_Trigger1:= Dry_Cycle OR (Cycle_Complete  AND NOT Enable_Motion),
			Off_Trigger2:= TRUE,
			Disable_Faults:= Dry_Cycle OR (Weld_Robots_WorkingOK) OR Turntable_Bypassed,
			Fault_Delay:= T#1.5s,
			Status=> Part_Present8,
			Faulted=>  PPFaults.8);

	(*Part 9 Present*)
		Part_Present9FB(
			Sensor_Input:= N02.I.0,
			On_Trigger1:= Enable_Motion AND In_Auto AND NOT Unload_Complete AND ((Model_ID=2) OR (Model_ID>=4)) AND NOT Welding_Complete ,
			On_Trigger2:= Model_ID>2,
			Off_Trigger1:= Dry_Cycle OR (Cycle_Complete  AND NOT Enable_Motion),
			Off_Trigger2:= TRUE,
			Disable_Faults:= Dry_Cycle OR (Weld_Robots_WorkingOK) OR Turntable_Bypassed,
			Fault_Delay:= T#1.5s,
			Status=> Part_Present9,
			Faulted=>  PPFaults.9);

	(*Part 10 Present*)
		Part_Present10FB(
			Sensor_Input:= N02.I.1,
			On_Trigger1:= Enable_Motion AND In_Auto AND NOT Unload_Complete AND (Model_ID>=4) AND NOT Welding_Complete ,
			On_Trigger2:= Model_ID>3,
			Off_Trigger1:= Dry_Cycle OR (Cycle_Complete  AND NOT Enable_Motion),
			Off_Trigger2:= TRUE,
			Disable_Faults:= Dry_Cycle OR (Weld_Robots_WorkingOK) OR Turntable_Bypassed,
			Fault_Delay:= T#1.5s,
			Status=> Part_Present10,
			Faulted=>  PPFaults.10);

	(*Part 11 Present*)
		Part_Present11FB(
			Sensor_Input:= N02.I.2,
			On_Trigger1:= Enable_Motion AND In_Auto AND NOT Unload_Complete AND (Model_ID>=5) AND NOT Welding_Complete ,
			On_Trigger2:= Model_ID>4,
			Off_Trigger1:= Dry_Cycle OR (Cycle_Complete  AND NOT Enable_Motion),
			Off_Trigger2:= TRUE,
			Disable_Faults:= Dry_Cycle OR (Weld_Robots_WorkingOK) OR Turntable_Bypassed,
			Fault_Delay:= T#1.5s,
			Status=> Part_Present11,
			Faulted=>  PPFaults.11);

	(*Part 12 Present*)
		Part_Present12FB(
			Sensor_Input:=  N02.I.3,
			On_Trigger1:= Enable_Motion AND In_Auto AND NOT Unload_Complete AND (Model_ID>=6) AND NOT Welding_Complete ,
			On_Trigger2:= Model_ID>5,
			Off_Trigger1:= Dry_Cycle OR (Cycle_Complete  AND NOT Enable_Motion),
			Off_Trigger2:= TRUE,
			Disable_Faults:= Dry_Cycle OR (Weld_Robots_WorkingOK) OR Turntable_Bypassed,
			Fault_Delay:= T#1.5s,
			Status=> Part_Present12,
			Faulted=>  PPFaults.12);

	(*Part 13 Present*)
		Part_Present13FB(
			Sensor_Input:= N02.I.4,
			On_Trigger1:= Enable_Motion AND In_Auto AND NOT Unload_Complete AND (Model_ID=7) AND NOT Welding_Complete ,
			On_Trigger2:= Model_ID>6,
			Off_Trigger1:= Dry_Cycle OR (Cycle_Complete  AND NOT Enable_Motion),
			Off_Trigger2:= TRUE,
			Disable_Faults:= Dry_Cycle OR (Weld_Robots_WorkingOK) OR Turntable_Bypassed,
			Fault_Delay:= T#1.5s,
			Status=> Part_Present13,
			Faulted=>  PPFaults.13);

	(*Part 14 Present*)
		Part_Present14FB(
			Sensor_Input:= N02.I.5,
			On_Trigger1:= Enable_Motion AND In_Auto AND NOT Unload_Complete AND (Model_ID=3) AND NOT Repo_Ack.0,
			On_Trigger2:= TRUE,
			Off_Trigger1:= Dry_Cycle OR (Cycle_Complete AND NOT Enable_Motion) OR Repo_Ack.0,
			Off_Trigger2:= TRUE,
			Disable_Faults:= Dry_Cycle OR (Weld_Robots_WorkingOK) OR Turntable_Bypassed,
			Fault_Delay:= T#1.5s,
			Status=> Part_Present14,
			Faulted=>  PPFaults.14);


	(*Part 15 Present*)
		Part_Present15FB(
			Sensor_Input:= N02.I.6,
			On_Trigger1:= Enable_Motion AND In_Auto AND NOT Unload_Complete,
			On_Trigger2:= NOT Repo_Reqs.0,
			Off_Trigger1:= Dry_Cycle OR (Cycle_Complete AND NOT Enable_Motion) OR Repo_Reqs.0,
			Off_Trigger2:= TRUE,
			Disable_Faults:= Dry_Cycle OR (Weld_Robots_WorkingOK) OR Turntable_Bypassed,
			Fault_Delay:= T#1.5s,
			Status=> Part_Present15,
			Faulted=>  PPFaults.15);

	(*Part 16 Present*)
		Part_Present16FB(
			Sensor_Input:= N02.I.7,
			On_Trigger1:= Enable_Motion AND In_Auto AND NOT Unload_Complete AND (Model_ID>=4) AND NOT Welding_Complete ,
			On_Trigger2:= TRUE,
			Off_Trigger1:= Dry_Cycle OR (Cycle_Complete  AND NOT Enable_Motion),
			Off_Trigger2:= TRUE,
			Disable_Faults:= Dry_Cycle OR (Weld_Robots_WorkingOK) OR Turntable_Bypassed,
			Fault_Delay:= T#1.5s,
			Status=> Part_Present16,
			Faulted=>  PPFaults.16);

	(*Part 17 Present*)
		Part_Present17FB(
			Sensor_Input:= N03.I.0,
			On_Trigger1:= Enable_Motion AND In_Auto AND NOT Unload_Complete AND (Model_ID>=5) AND NOT Welding_Complete ,
			On_Trigger2:= TRUE,
			Off_Trigger1:= Dry_Cycle OR (Cycle_Complete  AND NOT Enable_Motion),
			Off_Trigger2:= TRUE,
			Disable_Faults:= Dry_Cycle OR (Weld_Robots_WorkingOK) OR Turntable_Bypassed,
			Fault_Delay:= T#1.5s,
			Status=> Part_Present17,
			Faulted=>  PPFaults.17);

	(*Part 18 Present*)
		Part_Present18FB(
			Sensor_Input:= N03.I.1,
			On_Trigger1:= Enable_Motion AND In_Auto AND NOT Unload_Complete AND (Model_ID>=6) AND NOT Welding_Complete ,
			On_Trigger2:= TRUE,
			Off_Trigger1:= Dry_Cycle OR (Cycle_Complete  AND NOT Enable_Motion),
			Off_Trigger2:= TRUE,
			Disable_Faults:= Dry_Cycle OR (Weld_Robots_WorkingOK) OR Turntable_Bypassed,
			Fault_Delay:= T#1.5s,
			Status=> Part_Present18,
			Faulted=>  PPFaults.18);

	(*Part 19 Present*)
		Part_Present19FB(
			Sensor_Input:= N03.I.2,
			On_Trigger1:= Enable_Motion AND In_Auto AND NOT Unload_Complete AND (Model_ID=7) AND NOT Welding_Complete ,
			On_Trigger2:= TRUE,
			Off_Trigger1:= Dry_Cycle OR (Cycle_Complete  AND NOT Enable_Motion),
			Off_Trigger2:= TRUE,
			Disable_Faults:= Dry_Cycle OR (Weld_Robots_WorkingOK) OR Turntable_Bypassed,
			Fault_Delay:= T#1.5s,
			Status=> Part_Present19,
			Faulted=>  PPFaults.19);

	(*Part 20 Present*)
		Part_Present20FB(
			Sensor_Input:= N03.I.3,
			On_Trigger1:= Enable_Motion AND In_Auto AND NOT Welding_Complete AND (Model_ID<>3) AND NOT Welding_Complete ,
			On_Trigger2:= TRUE,
			Off_Trigger1:= Dry_Cycle OR (Cycle_Complete  AND NOT Enable_Motion),
			Off_Trigger2:= TRUE,
			Disable_Faults:= Dry_Cycle OR (Weld_Robots_WorkingOK) OR Turntable_Bypassed,
			Fault_Delay:= T#1.5s,
			Status=> Part_Present20,
			Faulted=>  PPFaults.20);

	(*Part 21 Present*)
		Part_Present21FB(
			Sensor_Input:= N03.I.4,
			On_Trigger1:= Enable_Motion AND In_Auto AND NOT Unload_Complete AND NOT Welding_Complete ,
			On_Trigger2:= (Model_ID =4) OR (Model_ID=11) OR (Model_ID=19) OR (Model_ID =5) OR (Model_ID=12) OR (Model_ID=20)
					   OR (Model_ID=6) OR (Model_ID=13) OR (Model_ID=21) OR (Model_ID=7) OR (Model_ID=14) OR (Model_ID=22),
			Off_Trigger1:= Dry_Cycle OR (Cycle_Complete  AND NOT Enable_Motion),
			Off_Trigger2:= TRUE,
			Disable_Faults:= Dry_Cycle OR (Weld_Robots_WorkingOK) OR Turntable_Bypassed,
			Fault_Delay:= T#1.5s,
			Status=> Part_Present21,
			Faulted=>  PPFaults.21);

	(*Part 22 Present*)
		Part_Present22FB(
			Sensor_Input:= N03.I.5,
			On_Trigger1:= Enable_Motion AND In_Auto AND NOT Unload_Complete,
			On_Trigger2:= NOT Repo_Reqs.0,
			Off_Trigger1:= Dry_Cycle OR (Cycle_Complete  AND NOT Enable_Motion) OR Repo_Reqs.0,
			Off_Trigger2:= TRUE,
			Disable_Faults:= Dry_Cycle OR (Weld_Robots_WorkingOK) OR Turntable_Bypassed,
			Fault_Delay:= T#1.5s,
			Status=> Part_Present22,
			Faulted=>  PPFaults.22);

	(*Part 23 Present*)
		Part_Present23FB(
			Sensor_Input:= N03.I.6,
			On_Trigger1:= Enable_Motion AND In_Auto AND NOT Unload_Complete,
			On_Trigger2:= NOT Repo_Reqs.0,
			Off_Trigger1:= Dry_Cycle OR (Cycle_Complete  AND NOT Enable_Motion) OR Repo_Reqs.0,
			Off_Trigger2:= TRUE,
			Disable_Faults:= Dry_Cycle OR (Weld_Robots_WorkingOK) OR Turntable_Bypassed,
			Fault_Delay:= T#1.5s,
			Status=> Part_Present23,
			Faulted=>  PPFaults.23);

	(*Part 24 Present*)
		Part_Present24FB(
			Sensor_Input:= N03.I.7,
			On_Trigger1:= Enable_Motion AND In_Auto AND NOT Unload_Complete AND (Model_ID<>3),
			On_Trigger2:= NOT Repo_Reqs.0,
			Off_Trigger1:= Dry_Cycle OR (Cycle_Complete  AND NOT Enable_Motion) OR Repo_Reqs.0,
			Off_Trigger2:= TRUE,
			Disable_Faults:= Dry_Cycle OR (Weld_Robots_WorkingOK) OR Turntable_Bypassed,
			Fault_Delay:= T#1.5s,
			Status=> Part_Present24,
			Faulted=>  PPFaults.24);

	(*Part 25 Present*)
		Part_Present25FB(
			Sensor_Input:= N04.I.0,
			On_Trigger1:= Enable_Motion AND In_Auto AND NOT Welding_Complete,
			On_Trigger2:= NOT Repo_Reqs.0,
			Off_Trigger1:= Dry_Cycle OR (Cycle_Complete  AND NOT Enable_Motion) OR Repo_Reqs.0,
			Off_Trigger2:= TRUE,
			Disable_Faults:= Dry_Cycle OR (Weld_Robots_WorkingOK) OR Turntable_Bypassed,
			Fault_Delay:= T#1.5s,
			Status=> Part_Present25,
			Faulted=>  PPFaults.25);

	(*Part 26 Present*)
		Part_Present26FB(
			Sensor_Input:= N04.I.1,
			On_Trigger1:= Enable_Motion AND In_Auto AND NOT Unload_Complete AND (Model_ID=3) AND NOT Repo_Ack.0,
			On_Trigger2:= TRUE,
			Off_Trigger1:= Dry_Cycle OR (Cycle_Complete  AND NOT Enable_Motion) OR Repo_Ack.0,
			Off_Trigger2:= TRUE,
			Disable_Faults:= Dry_Cycle OR (Weld_Robots_WorkingOK) OR Turntable_Bypassed,
			Fault_Delay:= T#1.5s,
			Status=> Part_Present26,
			Faulted=>  PPFaults.26);

	(*Part 27 Present*)
		Part_Present27FB(
			Sensor_Input:= N04.I.2,
			On_Trigger1:= Enable_Motion AND In_Auto AND NOT Welding_Complete AND (Model_ID<=2) AND NOT Welding_Complete ,
			On_Trigger2:= TRUE,
			Off_Trigger1:= Dry_Cycle OR (Cycle_Complete  AND NOT Enable_Motion),
			Off_Trigger2:= TRUE,
			Disable_Faults:= Dry_Cycle OR (Weld_Robots_WorkingOK) OR Turntable_Bypassed,
			Status=> Part_Present27,
			Faulted=>  PPFaults.27);

	(*Part 28 Present*)
		Part_Present28FB(
			Sensor_Input:= N04.I.3,
			On_Trigger1:= Enable_Motion AND In_Auto AND NOT Unload_Complete AND (Model_ID=2 AND NOT Welding_Complete),
			On_Trigger2:= TRUE,
			Off_Trigger1:= Dry_Cycle OR (Cycle_Complete  AND NOT Enable_Motion),
			Off_Trigger2:= TRUE,
			Disable_Faults:= Dry_Cycle OR (Weld_Robots_WorkingOK) OR Turntable_Bypassed,
			Fault_Delay:= T#1.5s,
			Status=> Part_Present28,
			Faulted=>  PPFaults.28);


	(*Part 29 Present*)
		Part_Present29FB(
			Sensor_Input:= N04.I.4,
			On_Trigger1:= Enable_Motion AND In_Auto AND NOT Unload_Complete AND (Model_ID>=4) AND NOT Welding_Complete ,
			On_Trigger2:= TRUE,
			Off_Trigger1:= Dry_Cycle OR (Cycle_Complete  AND NOT Enable_Motion),
			Off_Trigger2:= TRUE,
			Disable_Faults:= Dry_Cycle OR (Weld_Robots_WorkingOK) OR Turntable_Bypassed,
			Fault_Delay:= T#1.5s,
			Status=> Part_Present29,
			Faulted=>  PPFaults1.0);

	(*Part 30 Present*)
		Part_Present30FB(
			Sensor_Input:=N04.I.5,
			On_Trigger1:= Enable_Motion AND In_Auto AND NOT Unload_Complete AND (Model_ID>=5) AND NOT Welding_Complete ,
			On_Trigger2:= TRUE,
			Off_Trigger1:= Dry_Cycle OR (Cycle_Complete  AND NOT Enable_Motion),
			Off_Trigger2:= TRUE,
			Disable_Faults:= Dry_Cycle OR (Weld_Robots_WorkingOK) OR Turntable_Bypassed,
			Fault_Delay:= T#1.5s,
			Status=> Part_Present30,
			Faulted=>  PPFaults1.1);

	(*Part 31 Present*)
		Part_Present31FB(
			Sensor_Input:= N04.I.6,
			On_Trigger1:= Enable_Motion AND In_Auto AND NOT Unload_Complete AND (Model_ID>=6) AND NOT Welding_Complete ,
			On_Trigger2:= TRUE,
			Off_Trigger1:= Dry_Cycle OR (Cycle_Complete  AND NOT Enable_Motion),
			Off_Trigger2:= TRUE,
			Disable_Faults:= Dry_Cycle OR (Weld_Robots_WorkingOK) OR Turntable_Bypassed,
			Fault_Delay:= T#1.5s,
			Status=> Part_Present31,
			Faulted=>  PPFaults1.2);

	(*Part 32 Present*)
		Part_Present32FB(
			Sensor_Input:= N04.I.7,
			On_Trigger1:= Enable_Motion AND In_Auto AND NOT Unload_Complete AND (Model_ID=7) AND NOT Welding_Complete ,
			On_Trigger2:= TRUE,
			Off_Trigger1:= Dry_Cycle OR (Cycle_Complete  AND NOT Enable_Motion),
			Off_Trigger2:= TRUE,
			Disable_Faults:= Dry_Cycle OR (Weld_Robots_WorkingOK) OR Turntable_Bypassed,
			Fault_Delay:= T#1.5s,
			Status=> Part_Present32,
			Faulted=>  PPFaults1.3);

	(*Part 33 Present*)
		Part_Present33FB(
			Sensor_Input:= N05.I.0,
			On_Trigger1:= Enable_Motion AND In_Auto AND NOT Unload_Complete AND (Model_ID=7),
			On_Trigger2:= (Model_ID=7) OR (Model_ID=18) OR (Model_ID=22),
			Off_Trigger1:= Dry_Cycle OR (Cycle_Complete  AND NOT Enable_Motion),
			Off_Trigger2:= TRUE,
			Disable_Faults:= Dry_Cycle OR (Weld_Robots_WorkingOK) OR Turntable_Bypassed,
			Fault_Delay:= T#1.5s,
			Status=> Part_Present33,
			Faulted=>  PPFaults1.4);

	(*Part 34 Present*)
		Part_Present34FB(
			Sensor_Input:= N05.I.1,
			On_Trigger1:= Enable_Motion AND In_Auto AND NOT Unload_Complete,
			On_Trigger2:= (Model_ID=6) OR (Model_ID=17) OR (Model_ID=21) OR (Model_ID=7) OR (Model_ID=18) OR (Model_ID=22),
			Off_Trigger1:= Dry_Cycle OR (Cycle_Complete  AND NOT Enable_Motion),
			Off_Trigger2:= TRUE,
			Disable_Faults:= Dry_Cycle OR (Weld_Robots_WorkingOK) OR Turntable_Bypassed,
			Fault_Delay:= T#1.5s,
			Status=> Part_Present34,
			Faulted=>  PPFaults1.5);

	(*Part 35 Present*)
		Part_Present35FB(
			Sensor_Input:= N05.I.2,
			On_Trigger1:= Enable_Motion AND In_Auto AND NOT Unload_Complete,
			On_Trigger2:= (Model_ID =5) OR (Model_ID=16) OR (Model_ID=20)
					   OR (Model_ID=6) OR (Model_ID=17) OR (Model_ID=21) OR (Model_ID=7) OR (Model_ID=18) OR (Model_ID=22),
			Off_Trigger1:= Dry_Cycle OR (Cycle_Complete  AND NOT Enable_Motion),
			Off_Trigger2:= TRUE,
			Disable_Faults:= Dry_Cycle OR (Weld_Robots_WorkingOK) OR Turntable_Bypassed,
			Fault_Delay:= T#1.5s,
			Status=> Part_Present35,
			Faulted=>  PPFaults1.6);

	(*Part 36 Present*)
		Part_Present36FB(
			Sensor_Input:= N05.I.3,
			On_Trigger1:= Enable_Motion AND In_Auto AND NOT Unload_Complete,
			On_Trigger2:= (Model_ID =4) OR (Model_ID=15) OR (Model_ID=19) OR (Model_ID =5) OR (Model_ID=16) OR (Model_ID=20)
					   OR (Model_ID=6) OR (Model_ID=17) OR (Model_ID=21) OR (Model_ID=7) OR (Model_ID=18) OR (Model_ID=22),
			Off_Trigger1:= Dry_Cycle OR (Cycle_Complete  AND NOT Enable_Motion),
			Off_Trigger2:= TRUE,
			Disable_Faults:= Dry_Cycle OR (Weld_Robots_WorkingOK) OR Turntable_Bypassed,
			Fault_Delay:= T#1.5s,
			Status=> Part_Present36,
			Faulted=>  PPFaults1.7);

	(*Part 37 Present*)
		Part_Present37FB(
			Sensor_Input:= N05.I.4,
			On_Trigger1:= Enable_Motion AND In_Auto AND NOT Unload_Complete,
			On_Trigger2:= (Model_ID =4) OR (Model_ID=15) OR (Model_ID=19) OR (Model_ID =5) OR (Model_ID=16) OR (Model_ID=20)
					   OR (Model_ID=6) OR (Model_ID=17) OR (Model_ID=21) OR (Model_ID=7) OR (Model_ID=18) OR (Model_ID=22),
			Off_Trigger1:= Dry_Cycle OR (Cycle_Complete  AND NOT Enable_Motion),
			Off_Trigger2:= TRUE,
			Disable_Faults:= Dry_Cycle OR (Weld_Robots_WorkingOK) OR Turntable_Bypassed,
			Fault_Delay:= T#1.5s,
			Status=> Part_Present37,
			Faulted=>  PPFaults1.8);

	(*Part 38 Present*)
		Part_Present38FB(
			Sensor_Input:= N05.I.5,
			On_Trigger1:= Enable_Motion AND In_Auto AND NOT Unload_Complete,
			On_Trigger2:= NOT Repo_Reqs.0,
			Off_Trigger1:= Dry_Cycle OR (Cycle_Complete  AND NOT Enable_Motion) OR Repo_Reqs.0,
			Off_Trigger2:= TRUE,
			Disable_Faults:= Dry_Cycle OR (Weld_Robots_WorkingOK) OR Turntable_Bypassed,
			Fault_Delay:= T#1.5s,
			Status=> Part_Present38,
			Faulted=>  PPFaults1.9);

	(*Part 39 Present*)
		Part_Present39FB(
			Sensor_Input:= N05.I.6,
			On_Trigger1:= Enable_Motion AND In_Auto AND NOT Welding_Complete AND (Model_ID<>3),
			On_Trigger2:= TRUE,
			Off_Trigger1:= Dry_Cycle OR (Cycle_Complete  AND NOT Enable_Motion),
			Off_Trigger2:= TRUE,
			Disable_Faults:= Dry_Cycle OR (Weld_Robots_WorkingOK) OR Turntable_Bypassed,
			Fault_Delay:= T#1.5s,
			Status=> Part_Present39,
			Faulted=>  PPFaults1.10);

	(*Part 40 Present*)
		Part_Present40FB(
			Sensor_Input:= N05.I.7,
			On_Trigger1:= Enable_Motion AND In_Auto AND NOT Unload_Complete AND (Model_ID>=4) AND NOT Welding_Complete ,
			On_Trigger2:= TRUE,
			Off_Trigger1:= Dry_Cycle OR (Cycle_Complete  AND NOT Enable_Motion),
			Off_Trigger2:= TRUE,
			Disable_Faults:= Dry_Cycle OR (Weld_Robots_WorkingOK) OR Turntable_Bypassed,
			Fault_Delay:= T#1.5s,
			Status=> Part_Present40,
			Faulted=>  PPFaults1.11);

			
	(*Part 41 Present*)
		Part_Present41FB(
			Sensor_Input:= N06.I.0,
			On_Trigger1:= Enable_Motion AND In_Auto AND NOT Unload_Complete AND (Model_ID>=5) AND NOT Welding_Complete ,
			On_Trigger2:= TRUE,
			Off_Trigger1:= Dry_Cycle OR (Cycle_Complete  AND NOT Enable_Motion),
			Off_Trigger2:= TRUE,
			Disable_Faults:= Dry_Cycle OR (Weld_Robots_WorkingOK) OR Turntable_Bypassed,
			Fault_Delay:= T#1.5s,
			Status=> Part_Present41,
			Faulted=>  PPFaults1.12);

	(*Part 42 Present*)
		Part_Present42FB(
			Sensor_Input:= N06.I.1,
			On_Trigger1:= Enable_Motion AND In_Auto AND NOT Unload_Complete AND (Model_ID>=6) AND NOT Welding_Complete ,
			On_Trigger2:= TRUE,
			Off_Trigger1:= Dry_Cycle OR (Cycle_Complete  AND NOT Enable_Motion),
			Off_Trigger2:= TRUE,
			Disable_Faults:= Dry_Cycle OR (Weld_Robots_WorkingOK) OR Turntable_Bypassed,
			Fault_Delay:= T#1.5s,
			Status=> Part_Present42,
			Faulted=>  PPFaults1.13);

	(*Part 43 Present*)
		Part_Present43FB(
			Sensor_Input:= N06.I.2,
			On_Trigger1:= Enable_Motion AND In_Auto AND NOT Unload_Complete AND (Model_ID=7) AND NOT Welding_Complete ,
			On_Trigger2:= TRUE,
			Off_Trigger1:= Dry_Cycle OR (Cycle_Complete  AND NOT Enable_Motion),
			Off_Trigger2:= TRUE,
			Disable_Faults:= Dry_Cycle OR (Weld_Robots_WorkingOK) OR Turntable_Bypassed,
			Fault_Delay:= T#1.5s,
			Status=> Part_Present43,
			Faulted=>  PPFaults1.14);

	(*Part 44 Present*)
		Part_Present44FB(
			Sensor_Input:= N06.I.3,
			On_Trigger1:= Enable_Motion AND In_Auto AND NOT Unload_Complete AND (Model_ID=3) AND NOT Repo_Ack.0,
			On_Trigger2:= TRUE,
			Off_Trigger1:= Dry_Cycle OR (Cycle_Complete  AND NOT Enable_Motion) OR Repo_Ack.0,
			Off_Trigger2:= TRUE,
			Disable_Faults:= Dry_Cycle OR (Weld_Robots_WorkingOK) OR Turntable_Bypassed,
			Fault_Delay:= T#1.5s,
			Status=> Part_Present44,
			Faulted=>  PPFaults1.15);

	(*Part 45 Present*)
		Part_Present45FB(
			Sensor_Input:= N06.I.4,
			On_Trigger1:= Enable_Motion AND In_Auto AND NOT Unload_Complete,
			On_Trigger2:= (Model_ID=7) OR (Model_ID=14) OR (Model_ID=22),
			Off_Trigger1:= Dry_Cycle OR (Cycle_Complete  AND NOT Enable_Motion),
			Off_Trigger2:= TRUE,
			Disable_Faults:= Dry_Cycle OR (Weld_Robots_WorkingOK) OR Turntable_Bypassed,
			Fault_Delay:= T#1.5s,
			Status=> Part_Present45,
			Faulted=>  PPFaults1.16);

	(*Part 46 Present*)
		Part_Present46FB(
			Sensor_Input:= N06.I.5,
			On_Trigger1:= Enable_Motion AND In_Auto AND NOT Unload_Complete,
			On_Trigger2:= (Model_ID=6) OR (Model_ID=13) OR (Model_ID=21) OR (Model_ID=7) OR (Model_ID=14) OR (Model_ID=22),
			Off_Trigger1:= Dry_Cycle OR (Cycle_Complete  AND NOT Enable_Motion),
			Off_Trigger2:= TRUE,
			Disable_Faults:= Dry_Cycle OR (Weld_Robots_WorkingOK) OR Turntable_Bypassed,
			Fault_Delay:= T#1.5s,
			Status=> Part_Present46,
			Faulted=>  PPFaults1.17);

	(*Part 47 Present*)
		Part_Present47FB(
			Sensor_Input:= N06.I.6,
			On_Trigger1:= Enable_Motion AND In_Auto AND NOT Unload_Complete,
			On_Trigger2:= (Model_ID =5) OR (Model_ID=12) OR (Model_ID=20)
					   OR (Model_ID=6) OR (Model_ID=13) OR (Model_ID=21) OR (Model_ID=7) OR (Model_ID=14) OR (Model_ID=22),
			Off_Trigger1:= Dry_Cycle OR (Cycle_Complete  AND NOT Enable_Motion),
			Off_Trigger2:= TRUE,
			Disable_Faults:= Dry_Cycle OR (Weld_Robots_WorkingOK) OR Turntable_Bypassed,
			Fault_Delay:= T#1.5s,
			Status=> Part_Present47,
			Faulted=>  PPFaults1.18);

	(*Part 48 Present*)
		Part_Present48FB(
			Sensor_Input:= N06.I.7,
			On_Trigger1:= Enable_Motion AND In_Auto AND NOT Unload_Complete AND (Model_ID>=4),
			On_Trigger2:= (Model_ID =4) OR (Model_ID=11) OR (Model_ID=19) OR (Model_ID =5) OR (Model_ID=12) OR (Model_ID=20)
					   OR (Model_ID=6) OR (Model_ID=13) OR (Model_ID=21) OR (Model_ID=7) OR (Model_ID=14) OR (Model_ID=22),
			Off_Trigger1:= Dry_Cycle OR (Cycle_Complete  AND NOT Enable_Motion),
			Off_Trigger2:= TRUE,
			Disable_Faults:= Dry_Cycle OR (Weld_Robots_WorkingOK) OR Turntable_Bypassed,
			Fault_Delay:= T#1.5s,
			Status=> Part_Present48,
			Faulted=>  PPFaults1.19);

	(*Part 49 Present*)
		Part_Present49FB(
			Sensor_Input:= N07.I.0,
			On_Trigger1:= Enable_Motion AND In_Auto AND NOT Unload_Complete AND ((Model_ID<>3) OR (Model_ID<>10)),
			On_Trigger2:= (Model_ID =2) OR (Model_ID=9)
					   OR (Model_ID =4) OR (Model_ID=11) OR (Model_ID=19) OR (Model_ID =5) OR (Model_ID=12) OR (Model_ID=20)
					   OR (Model_ID=6) OR (Model_ID=13) OR (Model_ID=21) OR (Model_ID=7) OR (Model_ID=14) OR (Model_ID=22),
			Off_Trigger1:= Dry_Cycle OR (Cycle_Complete  AND NOT Enable_Motion),
			Off_Trigger2:= TRUE,
			Disable_Faults:= Dry_Cycle OR (Weld_Robots_WorkingOK) OR Turntable_Bypassed,
			Fault_Delay:= T#1.5s,
			Status=> Part_Present49,
			Faulted=>  PPFaults1.20);
			
	(*Part 50 Present*)
		Part_Present50FB(
			Sensor_Input:= N07.I.1,
			On_Trigger1:= Enable_Motion AND In_Auto AND NOT Unload_Complete AND (Model_ID<>3),
			On_Trigger2:= (Model_ID =1) OR (Model_ID=8) OR (Model_ID =2) OR (Model_ID=9)
					   OR (Model_ID =4) OR (Model_ID=11) OR (Model_ID=19) OR (Model_ID =5) OR (Model_ID=12) OR (Model_ID=20)
					   OR (Model_ID=6) OR (Model_ID=13) OR (Model_ID=21) OR (Model_ID=7) OR (Model_ID=14) OR (Model_ID=22),
			Off_Trigger1:= Dry_Cycle OR (Cycle_Complete  AND NOT Enable_Motion),
			Off_Trigger2:= TRUE,
			Disable_Faults:= Dry_Cycle OR (Weld_Robots_WorkingOK) OR Turntable_Bypassed,
			Fault_Delay:= T#1.5s,
			Status=> Part_Present50,
			Faulted=>  PPFaults1.21);			

	(*Part 51 Present*)
		Part_Present51FB(
			Sensor_Input:= N07.I.2,
			On_Trigger1:= Enable_Motion AND In_Auto AND NOT Unload_Complete,
			On_Trigger2:= TRUE,
			Off_Trigger1:= Dry_Cycle OR (Cycle_Complete  AND NOT Enable_Motion),
			Off_Trigger2:= TRUE,
			Disable_Faults:= Dry_Cycle OR (Weld_Robots_WorkingOK) OR Turntable_Bypassed,
			Fault_Delay:= T#1.5s,
			Status=> Part_Present51,
			Faulted=>  PPFaults1.22);

	(*Part 52 Present*)
		Part_Present52FB(
			Sensor_Input:= N07.I.3,
			On_Trigger1:= Enable_Motion AND In_Auto AND NOT Welding_Complete AND (Model_ID<>3),
			On_Trigger2:= TRUE,
			Off_Trigger1:= Dry_Cycle OR (Cycle_Complete  AND NOT Enable_Motion),
			Off_Trigger2:= TRUE,
			Disable_Faults:= Dry_Cycle OR (Weld_Robots_WorkingOK) OR Turntable_Bypassed,
			Fault_Delay:= T#1.5s,
			Status=> Part_Present52,
			Faulted=>  PPFaults1.23);

	(*Part 53 Present*)
		Part_Present53FB(
			Sensor_Input:= N07.I.4,
			On_Trigger1:= Enable_Motion AND In_Auto AND NOT Unload_Complete AND ((Model_ID=2 OR Model_ID>=4)AND NOT Welding_Complete),
			On_Trigger2:= TRUE,
			Off_Trigger1:= Dry_Cycle OR (Cycle_Complete  AND NOT Enable_Motion),
			Off_Trigger2:= TRUE,
			Disable_Faults:= Dry_Cycle OR (Weld_Robots_WorkingOK) OR Turntable_Bypassed,
			Fault_Delay:= T#1.5s,
			Status=> Part_Present53,
			Faulted=>  PPFaults1.24);

	(*Part 54 Present*)
		Part_Present54FB(
			Sensor_Input:= N07.I.5,
			On_Trigger1:= Enable_Motion AND In_Auto AND NOT Unload_Complete AND (Model_ID>=4) AND NOT Welding_Complete ,
			On_Trigger2:= TRUE,
			Off_Trigger1:= Dry_Cycle OR (Cycle_Complete  AND NOT Enable_Motion),
			Off_Trigger2:= TRUE,
			Disable_Faults:= Dry_Cycle OR (Weld_Robots_WorkingOK) OR Turntable_Bypassed,
			Fault_Delay:= T#1.5s,
			Status=> Part_Present54,
			Faulted=>  PPFaults1.25);

	(*Part 55 Present*)
		Part_Present55FB(
			Sensor_Input:= N07.I.6,
			On_Trigger1:= Enable_Motion AND In_Auto AND NOT Unload_Complete AND (Model_ID>=5) AND NOT Welding_Complete ,
			On_Trigger2:= TRUE,
			Off_Trigger1:= Dry_Cycle OR (Cycle_Complete  AND NOT Enable_Motion),
			Off_Trigger2:= TRUE,
			Disable_Faults:= Dry_Cycle OR (Weld_Robots_WorkingOK) OR Turntable_Bypassed,
			Fault_Delay:= T#1.5s,
			Status=> Part_Present55,
			Faulted=>  PPFaults1.26);

	(*Part 56 Present*)
		Part_Present56FB(
			Sensor_Input:= N07.I.7,
			On_Trigger1:= Enable_Motion AND In_Auto AND NOT Unload_Complete AND (Model_ID>=6) AND NOT Welding_Complete ,
			On_Trigger2:= TRUE,
			Off_Trigger1:= Dry_Cycle OR (Cycle_Complete  AND NOT Enable_Motion),
			Off_Trigger2:= TRUE,
			Disable_Faults:= Dry_Cycle OR (Weld_Robots_WorkingOK) OR Turntable_Bypassed,
			Fault_Delay:= T#1.5s,
			Status=> Part_Present56,
			Faulted=>  PPFaults1.27);

	(*Part 57 Present*)
		Part_Present57FB(
			Sensor_Input:= N08.I.0,
			On_Trigger1:= Enable_Motion AND In_Auto AND NOT Unload_Complete AND (Model_ID=7) AND NOT Welding_Complete ,
			On_Trigger2:= TRUE,
			Off_Trigger1:= Dry_Cycle OR (Cycle_Complete  AND NOT Enable_Motion),
			Off_Trigger2:= TRUE,
			Disable_Faults:= Dry_Cycle OR (Weld_Robots_WorkingOK) OR Turntable_Bypassed,
			Fault_Delay:= T#1.5s,
			Status=> Part_Present57,
			Faulted=>  PPFaults1.28);

	(*Part 72 Present*)
		Part_Present72FB(
			Sensor_Input:= N08.I.1,
			On_Trigger1:= Enable_Motion AND In_Auto AND (Model_ID=3) AND NOT Welding_Complete,
			On_Trigger2:= TRUE,
			Off_Trigger1:= Dry_Cycle OR (Cycle_Complete  AND NOT Enable_Motion) OR NOT (Model_ID=3),
			Off_Trigger2:= TRUE,
			Disable_Faults:= Dry_Cycle OR (Weld_Robots_WorkingOK) OR Turntable_Bypassed,
			Fault_Delay:= T#1.5s,
			Status=> Part_Present72,
			Faulted=>  PPFaults2.1);			
	
	(*Part 74 Present*)
		Part_Present74FB(
			Sensor_Input:= N08.I.2,
			On_Trigger1:= Enable_Motion AND In_Auto AND (Model_ID=3) AND NOT Welding_Complete,
			On_Trigger2:= TRUE,
			Off_Trigger1:= Dry_Cycle OR (Cycle_Complete  AND NOT Enable_Motion) OR NOT (Model_ID=3),
			Off_Trigger2:= TRUE,
			Disable_Faults:= Dry_Cycle OR (Weld_Robots_WorkingOK) OR Turntable_Bypassed,
			Fault_Delay:= T#1.5s,
			Status=> Part_Present74,
			Faulted=> PPFaults2.2);			
	
	(*Part 76 Present*)
		Part_Present76FB(
			Sensor_Input:= N08.I.3,
			On_Trigger1:= Enable_Motion AND In_Auto AND (Model_ID=3) AND NOT Welding_Complete,
			On_Trigger2:= TRUE,
			Off_Trigger1:= Dry_Cycle OR (Cycle_Complete  AND NOT Enable_Motion) OR NOT (Model_ID=3),
			Off_Trigger2:= TRUE,
			Disable_Faults:= Dry_Cycle OR (Weld_Robots_WorkingOK) OR Turntable_Bypassed,
			Fault_Delay:= T#1.5s,
			Status=> Part_Present76,
			Faulted=>  PPFaults2.3);		
	
	(*------------------- Sub Fixture Proxies -----------------------*)		
			
	(*--- Sub 42 - Model 504 and 542*)
	(*Part 58 Present*)
		Part_Present58FB(
			Sensor_Input:= N33.I.0,
			On_Trigger1:= Enable_Motion AND In_Auto AND NOT Unload_Complete AND (Model_ID=2),
			On_Trigger2:= TRUE,
			Off_Trigger1:= Dry_Cycle OR (Cycle_Complete  AND NOT Enable_Motion) OR (Model_ID=2 AND Repo_Ack.0),
			Off_Trigger2:= TRUE,
			Disable_Faults:= Dry_Cycle OR (Weld_Robots_WorkingOK) OR Turntable_Bypassed,
			Fault_Delay:= T#1.5s,
			Status=> Part_Present58,
			Faulted=>  PPFaults2.4);			

	(*Part 59 Present*)
		Part_Present59FB(
			Sensor_Input:= N33.I.1,
			On_Trigger1:= Enable_Motion AND In_Auto AND NOT Unload_Complete AND (Model_ID<=2),
			On_Trigger2:= TRUE,
			Off_Trigger1:= Dry_Cycle OR (Cycle_Complete  AND NOT Enable_Motion) OR (Model_ID<3 AND Repo_Ack.0),
			Off_Trigger2:= TRUE,
			Disable_Faults:= Dry_Cycle OR (Weld_Robots_WorkingOK) OR Turntable_Bypassed,
			Fault_Delay:= T#1.5s,
			Status=> Part_Present59,
			Faulted=>  PPFaults2.5);

	(*Part 60 Present*)
		Part_Present60FB(
			Sensor_Input:= N33.I.2,
			On_Trigger1:= Enable_Motion AND In_Auto AND NOT Unload_Complete AND (Model_ID=2),
			On_Trigger2:= TRUE,
			Off_Trigger1:= Dry_Cycle OR (Cycle_Complete  AND NOT Enable_Motion) OR (Model_ID<3 AND Repo_Ack.0),
			Off_Trigger2:= TRUE,
			Disable_Faults:= Dry_Cycle OR (Weld_Robots_WorkingOK) OR Turntable_Bypassed,
			Fault_Delay:= T#1.5s,
			Status=> Part_Present60,
			Faulted=>  PPFaults2.6);

	(*Part 61 Present*)
		Part_Present61FB(
			Sensor_Input:= N33.I.3,
			On_Trigger1:= Enable_Motion AND In_Auto AND NOT Unload_Complete AND (Model_ID=2),
			On_Trigger2:= TRUE,
			Off_Trigger1:= Dry_Cycle OR (Cycle_Complete  AND NOT Enable_Motion) OR (Model_ID<3 AND Repo_Ack.0),
			Off_Trigger2:= TRUE,
			Disable_Faults:= Dry_Cycle OR (Weld_Robots_WorkingOK) OR Turntable_Bypassed,
			Fault_Delay:= T#1.5s,
			Status=> Part_Present61,
			Faulted=>  PPFaults2.7);

	(*--- Sub 43 - Model 571*)
	(*Part 62 Present*)
		Part_Present62FB(
			Sensor_Input:= N35.I.0,
			On_Trigger1:= Enable_Motion AND In_Auto AND NOT Unload_Complete AND (Model_ID=7),
			On_Trigger2:= TRUE,
			Off_Trigger1:= Dry_Cycle OR (Cycle_Complete  AND NOT Enable_Motion) OR NOT (Model_ID=7),
			Off_Trigger2:= TRUE,
			Disable_Faults:= Dry_Cycle OR (Weld_Robots_WorkingOK) OR Turntable_Bypassed,
			Fault_Delay:= T#1.5s,
			Status=> Part_Present62,
			Faulted=>  PPFaults2.8);

	(*Part 63 Present*)
		Part_Present63FB(
			Sensor_Input:= N35.I.1,
			On_Trigger1:= Enable_Motion AND In_Auto AND NOT Unload_Complete AND (Model_ID=7),
			On_Trigger2:= TRUE,
			Off_Trigger1:= Dry_Cycle OR (Cycle_Complete  AND NOT Enable_Motion) OR NOT (Model_ID=7),
			Off_Trigger2:= TRUE,
			Disable_Faults:= Dry_Cycle OR (Weld_Robots_WorkingOK) OR Turntable_Bypassed,
			Fault_Delay:= T#1.5s,
			Status=> Part_Present63,
			Faulted=>  PPFaults2.9);

	(*Part 64 Present*)
		Part_Present64FB(
			Sensor_Input:= N35.I.2,
			On_Trigger1:= Enable_Motion AND In_Auto AND NOT Unload_Complete AND (Model_ID=7),
			On_Trigger2:= TRUE,
			Off_Trigger1:= Dry_Cycle OR (Cycle_Complete  AND NOT Enable_Motion) OR NOT (Model_ID=7),
			Off_Trigger2:= TRUE,
			Disable_Faults:= Dry_Cycle OR (Weld_Robots_WorkingOK) OR Turntable_Bypassed,
			Fault_Delay:= T#1.5s,
			Status=> Part_Present64,
			Faulted=>  PPFaults2.10);				

	(*--- Sub 44 - Model 550*)
	(*Part 65 Present*)
		Part_Present65FB(
			Sensor_Input:= N37.I.0,
			On_Trigger1:= Enable_Motion AND In_Auto AND NOT Unload_Complete AND (Model_ID=6),
			On_Trigger2:= TRUE,
			Off_Trigger1:= Dry_Cycle OR (Cycle_Complete  AND NOT Enable_Motion) OR NOT (Model_ID=6),
			Off_Trigger2:= TRUE,
			Disable_Faults:= Dry_Cycle OR (Weld_Robots_WorkingOK) OR Turntable_Bypassed,
			Fault_Delay:= T#1.5s,
			Status=> Part_Present65,
			Faulted=>  PPFaults2.11);

	(*Part 66 Present*)
		Part_Present66FB(
			Sensor_Input:= N37.I.1,
			On_Trigger1:= Enable_Motion AND In_Auto AND NOT Unload_Complete AND (Model_ID=6),
			On_Trigger2:= TRUE,
			Off_Trigger1:= Dry_Cycle OR (Cycle_Complete  AND NOT Enable_Motion) OR NOT (Model_ID=6),
			Off_Trigger2:= TRUE,
			Disable_Faults:= Dry_Cycle OR (Weld_Robots_WorkingOK) OR Turntable_Bypassed,
			Fault_Delay:= T#1.5s,
			Status=> Part_Present66,
			Faulted=>  PPFaults2.12);

	(*Part 67 Present*)
		Part_Present67FB(
			Sensor_Input:= N37.I.2,
			On_Trigger1:= Enable_Motion AND In_Auto AND NOT Unload_Complete AND (Model_ID=6),
			On_Trigger2:= TRUE,
			Off_Trigger1:= Dry_Cycle OR (Cycle_Complete  AND NOT Enable_Motion) OR NOT (Model_ID=6),
			Off_Trigger2:= TRUE,
			Disable_Faults:= Dry_Cycle OR (Weld_Robots_WorkingOK) OR Turntable_Bypassed,
			Fault_Delay:= T#1.5s,
			Status=> Part_Present67,
			Faulted=>  PPFaults2.13);

	(*--- Sub 45 - Model 536*)
	(*Part 68 Present*)
		Part_Present68FB(
			Sensor_Input:= N39.I.0,
			On_Trigger1:= Enable_Motion AND In_Auto AND NOT Unload_Complete AND (Model_ID=5),
			On_Trigger2:= TRUE,
			Off_Trigger1:= Dry_Cycle OR (Cycle_Complete  AND NOT Enable_Motion) OR NOT (Model_ID=5),
			Off_Trigger2:= TRUE,
			Disable_Faults:= Dry_Cycle OR (Weld_Robots_WorkingOK) OR Turntable_Bypassed,
			Fault_Delay:= T#1.5s,
			Status=> Part_Present68,
			Faulted=>  PPFaults2.14);

	(*Part 69 Present*)
		Part_Present69FB(
			Sensor_Input:= N39.I.1,
			On_Trigger1:= Enable_Motion AND In_Auto AND NOT Unload_Complete AND (Model_ID=5),
			On_Trigger2:= TRUE,
			Off_Trigger1:= Dry_Cycle OR (Cycle_Complete  AND NOT Enable_Motion) OR NOT (Model_ID=5),
			Off_Trigger2:= TRUE,
			Disable_Faults:= Dry_Cycle OR (Weld_Robots_WorkingOK) OR Turntable_Bypassed,
			Fault_Delay:= T#1.5s,
			Status=> Part_Present69,
			Faulted=>  PPFaults2.15);			

	(*--- Sub 46 - Model 526*)
	(*Part 70 Present*)
		Part_Present70FB(
			Sensor_Input:= N41.I.0,
			On_Trigger1:= Enable_Motion AND In_Auto AND NOT Unload_Complete AND (Model_ID=4),
			On_Trigger2:= TRUE,
			Off_Trigger1:= Dry_Cycle OR (Cycle_Complete  AND NOT Enable_Motion) OR NOT (Model_ID=4),
			Off_Trigger2:= TRUE,
			Disable_Faults:= Dry_Cycle OR (Weld_Robots_WorkingOK) OR Turntable_Bypassed,
			Fault_Delay:= T#1.5s,
			Status=> Part_Present70,
			Faulted=>  PPFaults2.16);			

	(*Part 71 Present*)
		Part_Present71FB(
			Sensor_Input:= N41.I.1,
			On_Trigger1:= Enable_Motion AND In_Auto AND NOT Unload_Complete AND (Model_ID=4),
			On_Trigger2:= TRUE,
			Off_Trigger1:= Dry_Cycle OR (Cycle_Complete  AND NOT Enable_Motion) OR NOT (Model_ID=4),
			Off_Trigger2:= TRUE,
			Disable_Faults:= Dry_Cycle OR (Weld_Robots_WorkingOK) OR Turntable_Bypassed,
			Fault_Delay:= T#1.5s,
			Status=> Part_Present71,
			Faulted=>  PPFaults2.17);			
			
	(*--- Sub 47 - Model 543*)
	(*Part 73 Present*)
		Part_Present73FB(
			Sensor_Input:= N43.I.0,
			On_Trigger1:= Enable_Motion AND In_Auto AND NOT Unload_Complete AND (Model_ID=3),
			On_Trigger2:= TRUE,
			Off_Trigger1:= Dry_Cycle OR (Cycle_Complete  AND NOT Enable_Motion) OR NOT (Model_ID=3),
			Off_Trigger2:= TRUE,
			Disable_Faults:= Dry_Cycle OR (Weld_Robots_WorkingOK) OR Turntable_Bypassed,
			Fault_Delay:= T#1.5s,
			Status=> Part_Present73,
			Faulted=>  PPFaults2.18);						
			
	(*Part 75 Present*)
		Part_Present75FB(
			Sensor_Input:= N43.I.1,
			On_Trigger1:= Enable_Motion AND In_Auto AND NOT Unload_Complete AND (Model_ID=3),
			On_Trigger2:= TRUE,
			Off_Trigger1:= Dry_Cycle OR (Cycle_Complete  AND NOT Enable_Motion) OR NOT (Model_ID=3),
			Off_Trigger2:= TRUE,
			Disable_Faults:= Dry_Cycle OR (Weld_Robots_WorkingOK) OR Turntable_Bypassed,
			Fault_Delay:= T#1.5s,
			Status=> Part_Present75,
			Faulted=>  PPFaults2.19);			
	
			

(*end*)
END_ACTION

ACTION Robot_Registration:


(*#################################### Register Robots to Tool ##################################*)
(*+++++++++++THIS AREA IS CUSTOM PER INSTALLATION AND WILL HAVE TO BE MODIFIED PER +++++++++++++*)
(*+++++++++++THIS AREA IS CUSTOM PER INSTALLATION AND WILL HAVE TO BE MODIFIED PER +++++++++++++*)
(*NOTE: See Example code in Fix 15 / 16*)
(*NOTE: See Example code in Fix 15 / 16*)

	(*Data From Load Robot(s)*)
	Load_Robots_Clear1:= TRUE;
	Load_Robots_Clear2:= TRUE;
	Load_Robots_Clear:=Load_Robots_Clear1 AND Load_Robots_Clear2;
	Load_Robots_WorkingOK1:= FALSE;
	Load_Robots_WorkingOK2:= FALSE;
	IF FALSE
		THEN
		Load_Robots_UnclampEarly1:= TRUE;
	END_IF;
	IF FALSE
		THEN
		Load_Robots_UnclampEarly2:= TRUE;
	END_IF;
	Load_Robots_Complete1:= FALSE;
	Load_Robots_Complete2:= FALSE;
	Load_Robots_PartInEOAT1:= FALSE;
	Load_Robots_PartInEOAT2:= FALSE;


	(*Data From Turntable*)
	TurntableA_Clear:= MAIN.R1.Clear_Of_HumanInterf1 AND NOT (MAIN.R1.Task_ID_Ack = Sweep_Fix01);
	TurntableB_Clear:= MAIN.R1.Clear_Of_HumanInterf2 AND NOT (MAIN.R1.Task_ID_Ack = Sweep_Fix02);
	Turntable_Clear:= TurntableA_Clear AND TurntableB_Clear;
	TurntableA_At_Robot:= (MAIN.R1.T03.I.0 AND MAIN.R1.T03.I.1);
	TurntableB_At_Robot:= (MAIN.R1.T03.I.2 AND MAIN.R1.T03.I.3);
	Turntable_WorkingOK:= ((MAIN.R1.Task_ID_Ack=Sweep_Fix02) AND MAIN.R1.At_HumanInterf2) OR ((MAIN.R1.Task_ID_Ack=Sweep_Fix01) AND MAIN.R1.At_HumanInterf1);
	TurntableA_Complete:= MAIN.R1.At_HumanInterf1 AND (MAIN.R1.Task_ID_Ack=Sweep_Fix01) AND MAIN.R1.Task_Completed;
	TurntableB_Complete:= MAIN.R1.At_HumanInterf2 AND (MAIN.R1.Task_ID_Ack=Sweep_Fix02) AND MAIN.R1.Task_Completed;


	(*Data From Seal Robot(s)*)
	Seal_Robots_Clear:= TRUE;
	Seal_Robots_WorkingOK:= FALSE;
	IF FALSE
		THEN
		Seal_Robots_UnclampEarly:= TRUE;
	END_IF;
	Seal_Robots_Complete:= FALSE;


	(*Data From Stud Robot(s)*)
	Stud_Robots_Clear:= TRUE;
	Stud_Robots_WorkingOK:= FALSE;
	IF FALSE
		THEN
		Stud_Robots_UnclampEarly:= TRUE;
	END_IF;
	Stud_Robots_Complete:= FALSE;


	(*Data From Weld Robot(s)*)
	Weld_Robots_Clear:= ((MAIN.R1.Clear_Of_EquipInterf1 AND NOT (MAIN.R1.Task_ID_Ack=Weld_Fix01) AND MAIN.R1.Clear_Of_EquipInterf8 AND NOT (MAIN.R1.Task_ID_Ack>=350)) OR MAIN.R1.At_Home)
					AND ((MAIN.R2.Clear_Of_EquipInterf1 AND NOT (MAIN.R2.Task_ID_Ack=Weld_Fix01) AND MAIN.R2.Clear_Of_EquipInterf8 AND NOT (MAIN.R2.Task_ID_Ack>=350)) OR MAIN.R2.At_Home)
					AND ((MAIN.R3.Clear_Of_EquipInterf1 AND NOT (MAIN.R3.Task_ID_Ack=Weld_Fix01) AND MAIN.R3.Clear_Of_EquipInterf8 AND NOT (MAIN.R3.Task_ID_Ack>=350)) OR MAIN.R3.At_Home);
					
	Weld_Robots_WorkingOK:= (MAIN.R1.Task_ID_Ack=Weld_Fix01) AND MAIN.R1.Operating
						AND (MAIN.R2.Task_ID_Ack=Weld_Fix01) AND MAIN.R2.Operating
						AND (MAIN.R3.Task_ID_Ack=Weld_Fix01) AND MAIN.R3.Operating;
						
	IF ((MAIN.R1.At_EquipInterf1 AND MAIN.R1.Clear_To_Unclamp AND NOT MAIN.R1.At_Pounce) 
		AND (MAIN.R2.At_EquipInterf1 AND MAIN.R2.Clear_To_Unclamp AND NOT MAIN.R2.At_Pounce)
		AND (MAIN.R3.At_EquipInterf1 AND MAIN.R3.Clear_To_Unclamp AND NOT MAIN.R3.At_Pounce))
		THEN
		Weld_Robots_UnclampEarly:= TRUE;
	END_IF;
	
	Weld_Robots_Complete:= (MAIN.R1.At_EquipInterf1 AND (MAIN.R1.Task_ID_Ack=Weld_Fix01) AND MAIN.R1.Task_Completed)
						AND (MAIN.R2.At_EquipInterf1 AND (MAIN.R2.Task_ID_Ack=Weld_Fix01) AND MAIN.R2.Task_Completed)
						AND (MAIN.R3.At_EquipInterf1 AND (MAIN.R3.Task_ID_Ack=Weld_Fix01) AND MAIN.R3.Task_Completed);
	
	(*Change Robots for Current Fixture functionality*) (*If no MIG robots Set to True.  Example code is in Fix15/16*) 
	Mig_Robots_Ready:=	((Main.R1.Fronius_Mig_HotKey AND Main.R2.Fronius_Mig_HotKey AND Main.R3.Fronius_Mig_Hotkey)
						AND (NOT Main.R1.Fronius_IgnitionError AND NOT Main.R2.Fronius_IgnitionError AND NOT Main.R3.Fronius_IgnitionError))
						OR (Dry_Cycle);
		
	

	(*Data From Unload Robot(s)*)
	Unload_Robots_Clear1:= ((MAIN.R4.Clear_Of_EquipInterf1 AND NOT (MAIN.R4.Task_ID_Ack=PickUp_Fix01)) OR MAIN.R4.At_Home);
	Unload_Robots_Clear2:= TRUE;
	Unload_Robots_Clear:= (Unload_Robots_Clear1 AND Unload_Robots_Clear2);
	Unload_Robots_WorkingOK1:= ((MAIN.R4.Task_ID_Ack=PickUp_Fix01) AND MAIN.R4.Operating);
	Unload_Robots_WorkingOK2:= FALSE;
	
	IF (MAIN.R4.At_EquipInterf1 AND MAIN.R4.Clear_To_Unclamp AND NOT MAIN.R4.At_Pounce)
		THEN
		Unload_Robots_UnclampEarly1:= TRUE;
	END_IF;
	IF FALSE
		THEN
		Unload_Robots_UnclampEarly1:= FALSE;
	END_IF;
	
	Unload_Robots_Complete1:= (MAIN.R4.At_EquipInterf1 AND (MAIN.R4.Task_ID_Ack=PickUp_Fix01) AND MAIN.R4.Task_Completed);
	Unload_Robots_Complete2:= FALSE;
	Unload_Robots_EOATEmpty1:= (EOAT04.EOAT_Part1_Empty);
	Unload_Robots_EOATEmpty2:= FALSE;




	(*Amalgumate All Robots Clear of Tool*)
	All_Robots_Clear:= Load_Robots_Clear AND Seal_Robots_Clear AND Stud_Robots_Clear AND Turntable_Clear AND Weld_Robots_Clear AND Unload_Robots_Clear;

	(*Data To All Robots*)
	(*Task ID*)
	R1_Data.Task_ID[1]:=Task_ID;
	R1_Data.Task_ID[9]:=Task_ID;
	R2_Data.Task_ID[9]:=Task_ID;
	R3_Data.Task_ID[9]:=Task_ID;
	R1_Data.Task_ID[11]:=Task_ID; (*THIS IS FOR WHEN R04 COMES FOR A PICK TO MOVE THE ROBOTS IN A PICK POSITION TLK*)
	R2_Data.Task_ID[11]:=Task_ID; (*THIS IS FOR WHEN R04 COMES FOR A PICK TO MOVE THE ROBOTS IN A PICK POSITION TLK*)
	R3_Data.Task_ID[11]:=Task_ID; (*THIS IS FOR WHEN R04 COMES FOR A PICK TO MOVE THE ROBOTS IN A PICK POSITION TLK*)
	IF TurnTableA_At_Robot THEN
	R4_Data.Task_ID[9]:=Task_ID;
	END_IF

	(*Fix ID*)
	R1_Data.Fix_ID[1]:=Fix_ID;
	R1_Data.Fix_ID[9]:=Fix_ID;
	R2_Data.Fix_ID[9]:=Fix_ID;
	R3_Data.Fix_ID[9]:=Fix_ID;
	R1_Data.Fix_ID[11]:=Fix_ID; (*THIS IS FOR WHEN R04 COMES FOR A PICK TO MOVE THE ROBOTS IN A PICK POSITION TLK*)
	R2_Data.Fix_ID[11]:=Fix_ID; (*THIS IS FOR WHEN R04 COMES FOR A PICK TO MOVE THE ROBOTS IN A PICK POSITION TLK*)
	R3_Data.Fix_ID[11]:=Fix_ID; (*THIS IS FOR WHEN R04 COMES FOR A PICK TO MOVE THE ROBOTS IN A PICK POSITION TLK*)
	IF TurnTableA_At_Robot THEN
	R4_Data.Fix_ID[9]:=Fix_ID;
	END_IF
	
	
	(*Model ID*)
	R1_Data.Model_ID[1]:=Model_ID;
	R1_Data.Model_ID[9]:=Model_ID;
	R2_Data.Model_ID[9]:=Model_ID;
	R3_Data.Model_ID[9]:=Model_ID;
	R1_Data.Model_ID[11]:=Model_ID; (*THIS IS FOR WHEN R04 COMES FOR A PICK TO MOVE THE ROBOTS IN A PICK POSITION TLK*)
	R2_Data.Model_ID[11]:=Model_ID; (*THIS IS FOR WHEN R04 COMES FOR A PICK TO MOVE THE ROBOTS IN A PICK POSITION TLK*)
	R3_Data.Model_ID[11]:=Model_ID; (*THIS IS FOR WHEN R04 COMES FOR A PICK TO MOVE THE ROBOTS IN A PICK POSITION TLK*)
	IF TurnTableA_At_Robot THEN
	R4_Data.Model_ID[9]:=Model_ID;
	END_IF

	(*Proceed from Pounce*)
	R1_Data.Proceed_From_Pounce[1]:= Robots_Clear_ToProceed;
	R1_Data.Proceed_From_Pounce[9]:= Robots_Clear_ToProceed;
	R2_Data.Proceed_From_Pounce[9]:= Robots_Clear_ToProceed;
	R3_Data.Proceed_From_Pounce[9]:= Robots_Clear_ToProceed;
	R1_Data.Proceed_From_Pounce[11]:= Robots_Clear_ToProceed; (*THIS IS FOR WHEN R04 COMES FOR A PICK TO MOVE THE ROBOTS IN A PICK POSITION TLK*)
	R2_Data.Proceed_From_Pounce[11]:= Robots_Clear_ToProceed; (*THIS IS FOR WHEN R04 COMES FOR A PICK TO MOVE THE ROBOTS IN A PICK POSITION TLK*)
	R3_Data.Proceed_From_Pounce[11]:= Robots_Clear_ToProceed; (*THIS IS FOR WHEN R04 COMES FOR A PICK TO MOVE THE ROBOTS IN A PICK POSITION TLK*)
	IF TurnTableA_At_Robot THEN
	R4_Data.Proceed_From_Pounce[9]:= Robots_Clear_ToProceed;
	END_IF

	(*Complete Acks*)
	R1_Data.Complete_Ack[1]:=(TurnA_Complete_Ack AND TurnTable_WorkingOK);
	R1_Data.Complete_Ack[9]:=(Weld_Complete_Ack AND Weld_Robots_WorkingOK);
	R2_Data.Complete_Ack[9]:=(Weld_Complete_Ack AND Weld_Robots_WorkingOK);
	R3_Data.Complete_Ack[9]:=(Weld_Complete_Ack AND Weld_Robots_WorkingOK);
	R1_Data.Complete_Ack[11]:=(Weld_Complete_Ack AND Weld_Robots_WorkingOK); (*THIS IS FOR WHEN R04 COMES FOR A PICK TO MOVE THE ROBOTS IN A PICK POSITION TLK*)
	R2_Data.Complete_Ack[11]:=(Weld_Complete_Ack AND Weld_Robots_WorkingOK); (*THIS IS FOR WHEN R04 COMES FOR A PICK TO MOVE THE ROBOTS IN A PICK POSITION TLK*)
	R3_Data.Complete_Ack[11]:=(Weld_Complete_Ack AND Weld_Robots_WorkingOK); (*THIS IS FOR WHEN R04 COMES FOR A PICK TO MOVE THE ROBOTS IN A PICK POSITION TLK*)
	IF TurnTableA_At_Robot THEN
	R4_Data.Complete_Ack[9]:=(Unload_Complete1_Ack AND Unload_Robots_WorkingOK1);
	END_IF

	(*Repo Acks*)
	R1_Data.PeripheralReq_Ack[9]:= Repo_Ack;
	R2_Data.PeripheralReq_Ack[9]:= Repo_Ack;
	R3_Data.PeripheralReq_Ack[9]:= Repo_Ack;
	R1_Data.PeripheralReq_Ack[11]:= Repo_Ack; (*THIS IS FOR WHEN R04 COMES FOR A PICK TO MOVE THE ROBOTS IN A PICK POSITION TLK*)
	R2_Data.PeripheralReq_Ack[11]:= Repo_Ack; (*THIS IS FOR WHEN R04 COMES FOR A PICK TO MOVE THE ROBOTS IN A PICK POSITION TLK*)
	R3_Data.PeripheralReq_Ack[11]:= Repo_Ack; (*THIS IS FOR WHEN R04 COMES FOR A PICK TO MOVE THE ROBOTS IN A PICK POSITION TLK*)
	IF TurnTableA_At_Robot THEN
	R4_Data.PeripheralReq_Ack[9]:= Repo_Ack;
	END_IF

